// TIA Portal V16 program export: 19 tag tables, 12 data types, 33 data blocks, 85 code blocks (in call order from the OBs), 112 instance data blocks

VAR_GLOBAL   // PLC tag table "Default tag table"
   System_Byte AT %MB1 : Byte;
   FirstScan AT %M1.0 : Bool;
   DiagStatusUpdate AT %M1.1 : Bool;
   AlwaysTRUE AT %M1.2 : Bool;
   AlwaysFALSE AT %M1.3 : Bool;
   Clock_Byte AT %MB2 : Byte;
   Clock_10Hz AT %M2.0 : Bool;
   Clock_5Hz AT %M2.1 : Bool;
   "Clock_2.5Hz" AT %M2.2 : Bool;
   Clock_2Hz AT %M2.3 : Bool;
   "Clock_1.25Hz" AT %M2.4 : Bool;
   Clock_1Hz AT %M2.5 : Bool;
   "Clock_0.625Hz" AT %M2.6 : Bool;
   "Clock_0.5Hz" AT %M2.7 : Bool;
   Byte_Wekt_DRV01_R AT %MB6 : SInt;   // Bytewejściowy Status napędu
   Byte_Wekt_DRV_Temp AT %MB7 : SInt;   // Byte temp pomocniczy przy wyliczeniu wektora
   "DRV01-Bit_A/M" AT %M6.7 : Bool;   // BIt IN statusu napędu Bit Aut/manual (aut=1, manu=0)
   "DRV01-Bit_REM" AT %M6.2 : Bool;   // Bit IN statusu napędu Bit-REM Tryb aut=1 rem=0 (REM sterowanie remontowe)
   "DRV01-Bit_A" AT %M6.0 : Bool;   // Bit IN status napędu Bit-A (Alarm)
   "DRV01-Bit_Z" AT %M6.5 : Bool;   // Bit IN statusu napędu Bit-Z rozkaz załącz
   "DRV01-Bit_W" AT %M6.4 : Bool;   // Bit IN status napędu Bit-W rozkaz wyłącz
   "DRV01-Bit_R" AT %M6.6 : Bool;   // Bit IN status napędu Bit-R sygnał RESET Alarmu
   Byte_Wekt_DRV01_L AT %MB8 : Byte;   // Byte OUT wektor napędu
   Bit_DRV01_A AT %M8.0 : Bool;   // Bit OUT wektor napędu Bit-A Alarm
   Bit_DRV01_REM AT %M8.2 : Bool;   // Bit OUT wektor napędu Bit-REM tryb pracy aut=1 rem=0 (REM-sterowanie remontowe)
   Bit_DRV01_Run AT %M8.3 : Bool;   // Bit OUT wektor napędu Bit-Run (Praca stycznik załączony)
   Bit_DRV01_W AT %M8.4 : Bool;   // Bit OUT wektor napędu Bit-W rozkaz wyłącz
   Bit_DRV01_Z AT %M8.5 : Bool;   // Bit OUT wektor napędu Bit-Z rozkaz załącz
   Bit_DRV01_R AT %M8.6 : Bool;   // Bit OUT wektor napędu Bit-R ( reset alarmu)
   "Bir_DRV01_A/M" AT %M8.7 : Bool;   // Bit OUT wektor napędu Bit-A/M rodzaj pracy auto / manual (aut=1, manu=0)
   Memeory_ResAut AT %M13.2 : Bool;   // Pamięć zbocza resetu bitu automat
   apx AT %MD28 : Real;
   apx1 AT %MD32 : Real;
   apy1 AT %MD24 : Real;
   osx AT %MD50 : Real;
   osx1 AT %MD54 : Real;
   osx2 AT %MD58 : Real;
   osy AT %MD62 : Real;
   osy1 AT %MD66 : Real;
   osy2 AT %MD70 : Real;
   State_PID1 AT %MW74 : Int;
   Error_State_PID1 AT %MD76 : DWord;
   SetpointLimit_H_PID1 AT %M14.0 : Bool;   // Wartość zadanaograniczenie górnego PID1
   SetpointLimit_L_PID1 AT %M14.1 : Bool;   // Wartość zadanaograniczenie dolnego PID1
   InputWarning_H_PID1 AT %M14.2 : Bool;   // Wejście ostrzegawcze progu górnrgo PID1
   InputWarning_L_PID1 AT %M14.3 : Bool;   // Wejście ostrzegawcze progu dolnego PID1
   Reset_PID1 AT %M14.4 : Bool;   // Znacznik resetu PID1
   My_1Hz AT %M206.7 : Bool;   // Generator 1hz
   memK1 AT %M15.1 : Bool;   // Flaga pamięci K1
   pause_1 AT %M15.4 : Bool;   // Dla pomiaru nr 1 funkcji FB3
   pause_2 AT %M15.5 : Bool;   // Pałza dla pomiaru nr 2 funkcji FB3
   "Q1.1" AT %Q1.1 : Bool;
   ProcessMemory_Static_1_setChanging AT %M206.4 : Bool;   // Znacznik pobierania konfiguracji do instancji pamięci peocesu
   Tag_2 AT %MW221 : Int;
   ResetPIDManual AT %M1100.0 : Bool;   // Ręczny reset PID
   Tag_5 AT %M10101.0 : Bool;
   Reset_symulowany AT %M1040.0 : Bool;   // Pomocniczy w razie symulacji
   Tag_6 AT %M1040.5 : Bool;
   Tag_7 AT %M1040.6 : Bool;
   Tag_8 AT %M1040.7 : Bool;
   ON_OFF_AQ_Falownik AT %M1040.2 : Bool;   // Do symulacji i testów
   Sumul_OnOFF_manual_PID AT %M1100.1 : Bool;
   Symula_K2_OFF_ONN AT %M1100.3 : Bool;   // Do testów
   ResetDodtkowe AT %M1100.6 : Bool;   // Potrzeby testowe
   SymulPomoc_04 AT %M1100.4 : Bool;
   SymulPomoc_05 AT %M1100.5 : Bool;
   "I0.0" AT %I0.0 : Bool;
   "Q0.0" AT %Q0.0 : Bool;
   "Q0.1" AT %Q0.1 : Bool;
   "Q0.2" AT %Q0.2 : Bool;
   "I0.1" AT %I0.1 : Bool;
   "I0.2" AT %I0.2 : Bool;
   "I0.5" AT %I0.5 : Bool;
   "I0.6" AT %I0.6 : Bool;
   "I0.7" AT %I0.7 : Bool;
   "I1.0" AT %I1.0 : Bool;
   "I1.1" AT %I1.1 : Bool;
   "I1.2" AT %I1.2 : Bool;
   "Q0.3" AT %Q0.3 : Bool;
   "Q0.4" AT %Q0.4 : Bool;
   "Q0.5" AT %Q0.5 : Bool;
   "I0.3" AT %I0.3 : Bool;
   "I0.4" AT %I0.4 : Bool;
   "I3.7" AT %I3.7 : Bool;
   "I1.3" AT %I1.3 : Bool;
   "I1.5" AT %I1.5 : Bool;
   "I2.1" AT %I2.1 : Bool;
   "I2.0" AT %I2.0 : Bool;
   "Q1.0" AT %Q1.0 : Bool;
   "Q2.3" AT %Q2.3 : Bool;
   "Q2.2" AT %Q2.2 : Bool;
   "I1.4" AT %I1.4 : Bool;
   "Q0.6" AT %Q0.6 : Bool;
   "Q0.7" AT %Q0.7 : Bool;
   "I2.2" AT %I2.2 : Bool;
   "I2.3" AT %I2.3 : Bool;
   "I2.4" AT %I2.4 : Bool;
   "I2.5" AT %I2.5 : Bool;
   "I2.6" AT %I2.6 : Bool;
   "I2.7" AT %I2.7 : Bool;
   "I3.0" AT %I3.0 : Bool;
   "I3.1" AT %I3.1 : Bool;
   "I3.2" AT %I3.2 : Bool;
   "I3.3" AT %I3.3 : Bool;
   "I3.4" AT %I3.4 : Bool;
   "I3.5" AT %I3.5 : Bool;
   "I3.6" AT %I3.6 : Bool;
   "Q2.0" AT %Q2.0 : Bool;
   "Q2.1" AT %Q2.1 : Bool;
   "Q2.4" AT %Q2.4 : Bool;
   "Q2.5" AT %Q2.5 : Bool;
   "Q2.6" AT %Q2.6 : Bool;
   "Q2.7" AT %Q2.7 : Bool;
   "Q3.0" AT %Q3.0 : Bool;
   "Q3.1" AT %Q3.1 : Bool;
   "Q3.2" AT %Q3.2 : Bool;
   "Q3.3" AT %Q3.3 : Bool;
   "Q3.4" AT %Q3.4 : Bool;
   "Q3.5" AT %Q3.5 : Bool;
   "Q3.6" AT %Q3.6 : Bool;
   "Q3.7" AT %Q3.7 : Bool;
   "I4.0" AT %I4.0 : Bool;
   "I4.1" AT %I4.1 : Bool;
   "I4.2" AT %I4.2 : Bool;
   "I4.3" AT %I4.3 : Bool;
   "I4.4" AT %I4.4 : Bool;
   "I4.5" AT %I4.5 : Bool;
   "I4.6" AT %I4.6 : Bool;
   "I4.7" AT %I4.7 : Bool;
   "Q4.0" AT %Q4.0 : Bool;
   "Q4.1" AT %Q4.1 : Bool;
   "Q4.2" AT %Q4.2 : Bool;
   "Q4.3" AT %Q4.3 : Bool;
   "Q4.4" AT %Q4.4 : Bool;
   "Q4.5" AT %Q4.5 : Bool;
   "Q4.6" AT %Q4.6 : Bool;
   "Q4.7" AT %Q4.7 : Bool;
   Tag_3 AT %MW410 : Int;
   Tag_4 AT %MW500 : Int;
   Tag_9 AT %MW502 : Int;
   Tag_10 AT %MD500 : DWord;
   ByteH_Status_P2 AT %MB24 : Byte;   // status napędu
   ByteH_Status_P3 AT %MB26 : Byte;   // staus napędu
   ByteH_Status_P4 AT %MB28 : Byte;   // status napędu
   activePump_P1 AT %M50.4 : Bool;   // aktywna w trybie automat
   activePump_P2 AT %M50.5 : Bool;   // aktywna w trybie automat
   activePump_P3 AT %M50.6 : Bool;   // aktywna w trybie automat
   activePump_P4 AT %M50.7 : Bool;   // aktywna w trybie automat
   PV_PER_bar_modbus AT %MW400 : Int;   // Wartość bar strefa 1
   increase_O2_no1 AT %M15.6 : Bool;   // Znacznik przyrostu wartości bar 1=przyrost, 0= brak przyrostu
   "PV_PER_bar_modbus(1)" AT %MW402 : Int;   // Wartość bar strefa 2
   Tag_1 AT %M212.3 : Bool;
   stopo_dodatkow_1 AT %M15.7 : Bool;   // wyłączenie dodatkowej 1
   ris1_Hz_Calkul_bar AT %M15.2 : Bool;   // Pamięć zbocza narastającego pomiaru 1 dla funkcji FB3
   ris2_Hz_Calkul_bar AT %M15.3 : Bool;   // Pamięć zbocza narastającego nr2 dla funkcji FB3
END_VAR
VAR_GLOBAL CONSTANT   // user constants
   CONST_BUFFER_OB82 : USInt := 200;
   CONST_CUREENT2TEMPERATURE_CONVERT : Real := 50.0;
   CONST_Hz_LEVEL : Real := 33.0;
   CONST_ADC_CONVERT : Real := 27648.0;
   CONST_OUTPUT_CAREENT : Real := 20.0;
   "Local~HSC_1(2)" : Hw_Hsc := 258;
   "Local~HSC_2(2)" : Hw_Hsc := 259;
   "Local~HSC_3(2)" : Hw_Hsc := 260;
   "Local~HSC_4(2)" : Hw_Hsc := 261;
   "Local~HSC_5(2)" : Hw_Hsc := 262;
   "Local~HSC_6(2)" : Hw_Hsc := 263;
   "Local~AI2_1" : Hw_SubModule := 264;
   "Local~DI14_DQ10_1" : Hw_SubModule := 265;
   "Local~Pulse_1(2)" : Hw_Pwm := 266;
   "Local~Pulse_2(2)" : Hw_Pwm := 267;
   "Local~Pulse_3(2)" : Hw_Pwm := 268;
   "Local~Pulse_4(2)" : Hw_Pwm := 269;
   DomZabkowska : DB_WWW := 333;
   Temeratura : DB_WWW := 333;
   "Local(2)" : Hw_SubModule := 50;
   "Local~PROFINET_interface_1(2)" : Hw_Interface := 64;
   "Local~PROFINET_interface_1~Port_1(2)" : Hw_Interface := 65;
   "Local~DI_8x24VDC_1(2)" : Hw_SubModule := 270;
   OB_Main : OB_PCYCLE := 1;
   "OB_Cyclic interrupt" : OB_Cyclic := 30;
   OB_Startup : OB_STARTUP := 100;
   "Local(1)" : Hw_SubModule := 50;
   "Local~PROFINET_interface_1(1)" : Hw_Interface := 64;
   "Local~PROFINET_interface_1~Port_1(1)" : Hw_Interface := 65;
   "Local~HSC_1(1)" : Hw_Hsc := 257;
   "Local~HSC_2(1)" : Hw_Hsc := 258;
   "Local~HSC_3(1)" : Hw_Hsc := 259;
   "Local~HSC_4(1)" : Hw_Hsc := 260;
   "Local~HSC_5(1)" : Hw_Hsc := 261;
   "Local~HSC_6(1)" : Hw_Hsc := 262;
   "Local~AI_2_AQ_2_1" : Hw_SubModule := 263;
   "Local~DI_14_DQ_10_1(1)" : Hw_SubModule := 264;
   "Local~Pulse_1(1)" : Hw_Pwm := 265;
   "Local~Pulse_2(1)" : Hw_Pwm := 266;
   "Local~Pulse_3(1)" : Hw_Pwm := 267;
   "Local~Pulse_4(1)" : Hw_Pwm := 268;
   "OB_Main(1)" : OB_PCYCLE := 1;
   "Local~DI_8x24VDC_1(1)" : Hw_SubModule := 269;
   "OB_Startup(1)" : OB_STARTUP := 100;
   "~Port_2" : Hw_Interface := 66;
   "Local~AQ_4x14BIT_1(1)" : Hw_SubModule := 271;
   "~Port_2(1)" : Hw_Interface := 66;
   MS_TO_S : DInt := 1000;
   MS_TO_M : DInt := 60000;   // Pomocnicza zmienna zamiana ms na minuty
END_VAR

VAR_GLOBAL   // PLC tag table "Analogs"
   IW68 AT %IW68 : Int;
   IW66 AT %IW66 : Int;
   IW64 AT %IW64 : Int;
   IW70 AT %IW70 : Int;
   switch_kolman AT %M18.7 : Bool;   // załącz/ wyłą filtrowanie przez kolmana analogów
   "i(1)" AT %MW112 : Int;
END_VAR

VAR_GLOBAL   // PLC tag table "Error"
   Led_Error AT %M17.5 : Bool;   // Znacznik sygnalizujący wystąpienie błędu sterownika Krat
   ResetErrorOB82 AT %M17.4 : Bool;   // Znacznik resetu licznika błędów
   alarmSuchobieg AT %M93.2 : Bool;   // bit alarmu wystąpienia suchobiegu pompownia
   alarmMagistrala_niskie_bar AT %M93.3 : Bool;   // bit alarmu wystąpienia btraku ciśnienia z magistrali
   "off_AlarmMagistrala-niskie_bar" AT %M93.4 : Bool;   // bit informuje o końcu awarii magistrali niskie
   alarm_max_bar_pompownia AT %M94.0 : Bool;   // bit alarmu przekroczono max bar pompownia B7
   Discrete_alarm_18 AT %M1025.1 : Bool;   // 16#0002: Niepoprawna wartość w parametrze "Input_PER". Sprawdź, czy na wejściu analogowym występuje błąd.
   "BitMeldun-7" AT %M1029.7 : Bool;   // 16#0080: Niepoprawna wartość w trybie pracy PID. Tryb pracy nie ulega zmianie.
   Discrete_alarm_13 AT %M1024.4 : Bool;   // 16#1000: Niepoprawna wartość w parametrze "Wartość zadana": Wartość nie ma prawidłowego formatu liczbowego.
   tmp_rezerwa_1 AT %M94.1 : Bool;   // bit rezerwowy 1
   bit_off_alarm_magistrala AT %M94.2 : Bool;   // ustaw jesli koniec alarmu na magistrali bar <min
END_VAR

VAR_GLOBAL   // PLC tag table "tags"
   "Tuning.TIR_visible" AT %M1002.0 : Bool;
   "Tuning.SUT_visible" AT %M1002.1 : Bool;
   "Tuning.Mode_visible" AT %M1002.2 : Bool;
   "PID_Compact.State" AT %MW1004 : Int;
   "PID_Compact.Setpoint" AT %MD1006 : Real;
   "PID_Compact.ScaledInput" AT %MD1010 : Real;
   "PID_Compact.Output_PWM" AT %M1014.0 : Bool;
   "PID_Compact.ModeActivate" AT %M1014.1 : Bool;
   "PID_Compact.ManualEnable" AT %M1014.2 : Bool;
   "PID_Compact.Disturbance" AT %MD1016 : Real;
   "HMI.Setpoint_limited" AT %M1020.0 : Bool;
   "HMI.PhysicalUnit" AT %MB1021 : Char;
   "HMI.Output_PWM_USInt" AT %MB1022 : USInt;
   "HMI.ManualMode_visible(1)" AT %M1023.0 : Bool;
   "HMI.ManualMode_visible" AT %M1023.1 : Bool;
   "HMI.ErrorBits_Int" AT %MW1024 : Int;
   "HMI.ErrorAck_Int" AT %MW1026 : Int;
   "HMI.Warning_Int" AT %MW1028 : Int;
   "HMI.ErrorAck" AT %M1030.0 : Bool;
   "HMI.Acknowledge_visible" AT %M1030.1 : Bool;
   Communication_Alarm AT %M1030.2 : Bool;   // Znacznik błedu komunikacji HMI - PLC
   outAlarm AT %M1030.3 : Bool;   // Znacznik alarmu zbiorczego (Sygnalizator)
   "HMI.alarm_byte_1" AT %MW800 : Word;   // słowo alarmów
   "HMI.gotowość_falownik_1" AT %M800.0 : Bool;   // gotowość falownika 1
   "HMI.brak_zasilania" AT %M800.1 : Bool;   // brak zasilnia
   "HMI.SłowoStatus_Falownik1" AT %MW2000 : Int;   // Słowo statusu falownika F1
   "HMI.FalSata_bit_0" AT %M2000.0 : Bool;   // Sterowanie poprawne
   "HMI.FalSata_bit_1" AT %M2000.1 : Bool;   // falownik gotowość
   "HMI.FalSata_bit_2" AT %M2000.2 : Bool;   // wybieg
   "HMI.FalSata_bit_3" AT %M2000.3 : Bool;   // trip error
   "HMI.FalSata_bit_4" AT %M2000.4 : Bool;   // no trip error
   "HMI.FalSata_bit_5" AT %M2000.5 : Bool;   // reserved
   "HMI.FalSata_bit_6" AT %M2000.6 : Bool;   // trip zablokowany
   "HMI.FalSata_bit_7" AT %M2000.7 : Bool;   // Ostrzeżenie
   "HMI.FalSata_bit_8" AT %M2001.0 : Bool;   // prędkość = referencyjnej
   "HMI.FalSata_bit_9" AT %M2001.1 : Bool;   // listwa sterowania
   "HMI.FalSata_bit_10" AT %M2001.2 : Bool;   // częstotliwość ok
   "HMI.FalSata_bit_11" AT %M2001.3 : Bool;   // praca
   "HMI.FalSata_bit_12" AT %M2001.4 : Bool;   // rezystor hamowania
   "HMI.FalSata_bit_13" AT %M2001.5 : Bool;   // volty przekroczone
   "HMI.FalSata_bit_14" AT %M2001.6 : Bool;   // problem z momentem obrotowym
   "HMI.FalSata_bit_15" AT %M2001.7 : Bool;   // zabezpieczenie termiczne
   "HMI.kasowanie.ekranów" AT %MW1000 : Int;
   "HMI.kasowanie.ekranów_bit_0" AT %M1000.0 : Bool;   // kasowanie alarmu ekran pomp
   "HMI.kasowanie.ekranów_bit_1" AT %M1000.1 : Bool;   // kasowanie alarmu ekran zasów
   "HMI.kasowanie.ekranów_bit_2" AT %M1000.2 : Bool;
   "HMI.kasowanie.ekranów_bit_3" AT %M1000.3 : Bool;
   "HMI.kasowanie.ekranów_bit_4" AT %M1000.4 : Bool;
   "HMI.kasowanie.ekranów_bit_5" AT %M1000.5 : Bool;
   "HMI.kasowanie.ekranów_bit_6" AT %M1000.6 : Bool;
   "HMI.kasowanie.ekranów_bit_7" AT %M1000.7 : Bool;
   "HMI.alarm_01" AT %M1001.0 : Bool;   // Alarm Modbus RTU
   "HMI.alarm_02" AT %M1001.1 : Bool;   // Ostrzerzenie Modbus RTU
   "HMI.alarm_01(2)" AT %M1001.2 : Bool;
   "HMI.alarm_01(3)" AT %M1001.3 : Bool;
   "HMI.alarm_01(4)" AT %M1001.4 : Bool;
   "HMI.alarm_01(5)" AT %M1001.5 : Bool;
   "HMI.alarm_01(6)" AT %M1001.6 : Bool;
   "HMI.alarm_01(7)" AT %M1001.7 : Bool;
END_VAR

VAR_GLOBAL   // PLC tag table "MP04_1"
   temp_current_fow_H_Q1 AT %MW600 : Word;   // H byte przepływ aktualny VF
   tmp_current_fow_L_Q1 AT %MW602 : Word;   // L byte przepływ aktualny VF
   tmp_front_volumeVF_H_Q1 AT %MW604 : Word;   // licznik objetości przód H byte
   tmp_front_volumeVF_L_Q1 AT %MW606 : Word;   // licznik objetości przód L byte
   tmp_back_balueVR_H_Q1 AT %MW608 : Word;   // licznik objętości wstecz H byte
   tmp_back_balueVR_L_Q1 AT %MW610 : Word;   // licznik objętości wstecz L byte
   "tmp_differential counter VD_H_Q1" AT %MW612 : Word;   // licznik różnicowy VD H byte
   "tmp_differential counter VD_L_Q1" AT %MW614 : Word;   // licznik różnicowy VD L byte
   "tmp_volume counter status _GF_H_Q1" AT %MW616 : Word;   // statu licznik objetości GF H byte
   "tmp_volume counter status _GF_L_Q1" AT %MW618 : Word;   // status licznik objetości GF L byte
   "tmp_volume counter status_GR_H_Q1" AT %MW620 : Word;   // statu licznik objetości GR H byte
   "tmp_volume counter status_GR_L_Q1" AT %MW622 : Word;   // statu licznik objetości GR L byte
   "tmp_differential counter status_GD_H_Q1" AT %MW624 : Word;   // statu licznik objetości GD H byte
   "tmp_differential counter status_GD_L_Q1" AT %MW626 : Word;   // statu licznik objetości GD L byte
   tmp_sataus_MP04_Q1 AT %MW628 : Word;   // staus urządzenia MP04_Q1
   temp_current_fow_H_Q2 AT %MW630 : Word;   // H byte przepływ aktualny VF
   tmp_current_fow_L_Q2 AT %MW632 : Word;   // L byte przepływ aktualny VF
   tmp_front_volumeVF_H_Q2 AT %MW634 : Word;   // licznik objetości przód H byte
   tmp_front_volumeVF_L_Q2 AT %MW636 : Word;   // licznik objetości przód L byte
   tmp_back_balueVR_H_Q2 AT %MW638 : Word;   // licznik objętości wstecz H byte
   tmp_back_balueVR_L_Q2 AT %MW640 : Word;   // licznik objętości wstecz L byte
   "tmp_differential counter VD_H_Q2" AT %MW642 : Word;   // licznik różnicowy VD H byte
   "tmp_differential counter VD_L_Q2" AT %MW644 : Word;   // licznik różnicowy VD L byte
   "tmp_volume counter status _GF_H_Q2" AT %MW646 : Word;   // statu licznik objetości GF H byte
   "tmp_volume counter status _GF_L_Q2" AT %MW648 : Word;   // status licznik objetości GF L byte
   "tmp_volume counter status_GR_H_Q2" AT %MW650 : Word;   // statu licznik objetości GR H byte
   "tmp_volume counter status_GR_L_Q2" AT %MW652 : Word;   // statu licznik objetości GR L byte
   "tmp_differential counter status_GD_H_Q2" AT %MW654 : Word;   // statu licznik objetości GD H byte
   "tmp_differential counter status_GD_L_Q2" AT %MW656 : Word;   // statu licznik objetości GD L byte
   tmp_sataus_MP04_Q2 AT %MW658 : Word;   // staus urządzenia MP04_Q2
END_VAR

VAR_GLOBAL   // PLC tag table "ModbusRTU"
   setErrorModbsmasterFal AT %M18.0 : Bool;   // error bit modbus master falownik / Znacznik błedu komunikacji modbus
   setErrorModbsmasterMPP04_1 AT %M18.1 : Bool;   // error bit modbus master przepływomierz / Znacznik błedu komunikacji modbus
   setErrorModbsSlave AT %M18.2 : Bool;   // error bit modbus slave / Znacznik błedu komunikacji modbus
   "setErrorModbs----" AT %M18.3 : Bool;   // Znacznik błedu komunikacji modbus
   memRisErrorModbusmaster AT %M16.6 : Bool;   // Pamięć zbocza błędu komunikacji
   memReisModbus_Loop1 AT %M16.2 : Bool;   // Znacznik pamięci zbocza dla pętli 1
   memRisModbusmaster_Loop2 AT %M16.3 : Bool;   // pamięć zbocza dla petli 2 modbas
   memRisModbusmaster_Loop3 AT %M16.4 : Bool;   // pamięć zbocza pętli 3 modbas
   memRisModbus_Loop AT %M16.5 : Bool;   // Pamieć zbocza do uruchomienia petli SC1000
   ndrSlave AT %M16.7 : Bool;   // bit nowe dane gotowe / Pamieć zbocza błedu komunikacji
   drSlave AT %M14.5 : Bool;   // bit czytanie danych / pamięć zbocza błędu komunikacji
   memRisErrorModbusMPP04_1 AT %M14.6 : Bool;   // pamięć zbocza error modbus MPP04-1
   StatusSlave AT %MW29 : Word;   // Status slave Modbus RTU
   errorSatausSlave AT %MW31 : Word;   // Status błędu slave Modbus RTU
   setErrorModbsmasterMPP04_2 AT %M93.0 : Bool;   // error bit modbus master przepływomierz / Znacznik błedu komunikacji modbus
   memRisErrorModbusMPP04_2 AT %M14.7 : Bool;   // pamięć zbocza error modbus MPP04-1
   memRisErrorModbusFal AT %M93.1 : Bool;   // pamięć zbocza error modbus MPP04-1
   "memStep_errorMPP04-1" AT %MB100 : USInt;   // bajt pamieci w którym kroku nastąpił błąd modbus
   "memStep_errorMPP04-2" AT %MB101 : USInt;   // bajt pamieci w którym kroku nastąpił błąd modbus
   memStep_errorFal AT %MB102 : USInt;   // bajt pamieci w którym kroku nastąpił błąd modbus
   memStep_errorSlave AT %MB103 : USInt;   // bajt pamieci w którym kroku nastąpił błąd modbus
   "memRisSteperror_MPP04-1" AT %M104.0 : Bool;   // pamięć zbocza dla przechwycenia kroku błedu
   "memRisSteperror_MPP04-2" AT %M104.1 : Bool;   // pamięć zbocza dla przechwycenia kroku błedu
   memRisSteperror_Fal AT %M104.2 : Bool;   // pamięć zbocza dla przechwycenia kroku błedu
   memRisSteperror AT %M104.3 : Bool;   // pamięć zbocza dla przechwycenia kroku błedu
   act_flow_Q1 AT %MD600 : DWord;   // wartość przepływu Q1
   act_front_volumeVF_Q1 AT %MD604 : DWord;   // licznik objetości przód Q1
   act_back_valueVR_Q1 AT %MD608 : DWord;   // licznika objętości w tył Q1
   "act_differential counter VD_Q1" AT %MD612 : DWord;   // liczni różnicowyobjętości VD Q1
   "act_volume counter status _GF_Q1" AT %MD616 : DWord;   // główny licznik objetosci przód GF Q1
   "act_volume counter status_GR_Q1" AT %MD620 : DWord;   // główny licznik objetości w tył GR Q1
   "act_differential counter status_GD_Q1" AT %MD624 : DWord;   // główny różnicow licznik objetości GD Q1
   act_flow_Q2 AT %MD630 : DWord;   // wartość przepływu Q2
   act_ValueVF_Q2 AT %MD634 : DWord;   // licznik objetości przód Q2
   act_front_volumeVF_Q2 AT %MD638 : DWord;   // licznika objętości w tył Q2
   act_back_balueVR_Q2 AT %MD642 : DWord;   // liczni różnicowyobjętości VD Q2
   "act_differential counter VD_Q2" AT %MD646 : DWord;   // główny licznik objetosci przód GF Q2
   "act_volume counter status _GF_Q2" AT %MD650 : DWord;   // główny licznik objetości w tył GR Q2
   "act_volume counter status_GR_Q2" AT %MD654 : DWord;   // główny różnicow licznik objetości GD Q2
   "act_differential counter status_GD_Q2" AT %MD658 : DWord;
   Switch_PrzepłtwSygnał AT %M92.0 : Bool;   // wybór źródła wartości pomiaru analog / modbus rtu
END_VAR

VAR_GLOBAL   // PLC tag table "ModbusTCP"
   memTrgServer_1 AT %M106.0 : Bool;
   memTrgServer_2 AT %M106.1 : Bool;
   memTrgServer_3 AT %M106.2 : Bool;
   DISCONNECT_SERVER_1 AT %M106.3 : Bool;
   DISCONNECT_SERVER_2 AT %M106.4 : Bool;
   DISCONNECT_SERVER_3 AT %M106.5 : Bool;
   memRisingTriger_Data_4 AT %M107.1 : Bool;   // pamieć zbocza narastającego przekazania danej do wysłania
   memRisingTriger_Data_11 AT %M108.0 : Bool;   // pamieć zbocza narastającego przekazania danej do wysłania
   memRisingTriger_Data_5 AT %M107.2 : Bool;   // pamieć zbocza narastającego przekazania danej do wysłania
   memRisingTriger_Data_8 AT %M107.5 : Bool;   // pamieć zbocza narastającego przekazania danej do wysłania
   memRisingTriger_Data_1 AT %M106.6 : Bool;   // pamieć zbocza narastającego przekazania danej do wysłania
   memRisingTriger_Data_13 AT %M108.2 : Bool;   // pamieć zbocza narastającego przekazania danej do wysłania
   memRisingTriger_Data_2 AT %M106.7 : Bool;   // pamieć zbocza narastającego przekazania danej do wysłania
   memRisingTriger_Data_6 AT %M107.3 : Bool;   // pamieć zbocza narastającego przekazania danej do wysłania
   memRisingTriger_Data_10 AT %M107.7 : Bool;   // pamieć zbocza narastającego przekazania danej do wysłania
   memRisingTriger_Data_12 AT %M108.1 : Bool;   // pamieć zbocza narastającego przekazania danej do wysłania
   memRisingTriger_Data_3 AT %M107.0 : Bool;   // pamieć zbocza narastającego przekazania danej do wysłania
   memRisingTriger_Data_9 AT %M107.6 : Bool;   // pamieć zbocza narastającego przekazania danej do wysłania
   memRisingTriger_Data_7 AT %M107.4 : Bool;   // pamieć zbocza narastającego przekazania danej do wysłania
   DISCONNECT_SERVER_4 AT %M108.3 : Bool;
   memTrgServer_4 AT %M108.4 : Bool;
   memTrig_Client_Receiving_16 AT %M110.4 : Bool;
   memTrig_Client_Receiving_7 AT %M109.3 : Bool;
   memTrig_Client_Receiving_11 AT %M109.7 : Bool;
   memRisingTriger_Data_1_2 AT %M110.6 : Bool;   // pamieć zbocza narastającego przekazania danej do wysłania
   memRisingTriger_Data_1_1 AT %M110.5 : Bool;   // pamieć zbocza narastającego przekazania danej do wysłania
   memTrig_Client_Receiving_5 AT %M109.1 : Bool;
   memTrig_Client_Receiving_13 AT %M110.1 : Bool;
   memTrig_Client_Receiving_14 AT %M110.2 : Bool;
   memTrig_Client_Receiving_3 AT %M108.7 : Bool;
   memTrig_Client_Receiving_8 AT %M109.4 : Bool;
   memTrig_Client_Receiving_10 AT %M109.6 : Bool;
   memTrig_Client_Receiving_6 AT %M109.2 : Bool;
   memTrig_Client_Receiving_12 AT %M110.0 : Bool;
   memTrig_Client_Receiving_2 AT %M108.6 : Bool;
   memTrig_Client_Receiving_1 AT %M108.5 : Bool;
   memTrig_Client_Receiving_4 AT %M109.0 : Bool;
   memTrig_Client_Receiving_9 AT %M109.5 : Bool;
   memTrig_Client_Receiving_15 AT %M110.3 : Bool;
   memRisingTriger_Data_16 AT %M111.2 : Bool;
   memRisingTriger_Data_14 AT %M111.0 : Bool;
   memRisingTriger_Data_15 AT %M111.1 : Bool;
   memRisingTriger_Data_47 AT %M115.1 : Bool;
   memTrig_Client_Receiving_17 AT %M120.2 : Bool;
   memTrig_Client_Receiving_87 AT %M129.0 : Bool;
   memTrig_Client_Receiving_23 AT %M121.0 : Bool;
   memRisingTriger_Data_29 AT %M112.7 : Bool;
   memTrig_Client_Receiving_84 AT %M128.5 : Bool;
   memTrig_Client_Receiving_43 AT %M123.4 : Bool;
   memRisingTriger_Data_63 AT %M117.1 : Bool;
   memTrig_Client_Receiving_74 AT %M127.3 : Bool;
   memRisingTriger_Data_69 AT %M117.7 : Bool;
   memRisingTriger_Data_70 AT %M118.0 : Bool;
   memTrig_Client_Receiving_32 AT %M122.1 : Bool;
   memRisingTriger_Data_80 AT %M119.2 : Bool;
   memTrig_Client_Receiving_65 AT %M126.2 : Bool;
   memTrig_Client_Receiving_71 AT %M127.0 : Bool;
   memTrig_Client_Receiving_36 AT %M122.5 : Bool;
   memRisingTriger_Data_84 AT %M119.6 : Bool;
   memRisingTriger_Data_68 AT %M117.6 : Bool;
   memTrig_Client_Receiving_49 AT %M124.2 : Bool;
   memRisingTriger_Data_85 AT %M119.7 : Bool;
   memRisingTriger_Data_36 AT %M113.6 : Bool;
   memTrig_Client_Receiving_76 AT %M127.5 : Bool;
   memTrig_Client_Receiving_70 AT %M126.7 : Bool;
   memTrig_Client_Receiving_89 AT %M129.2 : Bool;
   memRisingTriger_Data_19 AT %M111.5 : Bool;
   memRisingTriger_Data_31 AT %M113.1 : Bool;
   memTrig_Client_Receiving_20 AT %M120.5 : Bool;
   memTrig_Client_Receiving_48 AT %M124.1 : Bool;
   memTrig_Client_Receiving_56 AT %M125.1 : Bool;
   memRisingTriger_Data_44 AT %M114.6 : Bool;
   memTrig_Client_Receiving_82 AT %M128.3 : Bool;
   memTrig_Client_Receiving_58 AT %M125.3 : Bool;
   memTrig_Client_Receiving_67 AT %M126.4 : Bool;
   memRisingTriger_Data_57 AT %M116.3 : Bool;
   memTrig_Client_Receiving_80 AT %M128.1 : Bool;
   memRisingTriger_Data_52 AT %M115.6 : Bool;
   memTrig_Client_Receiving_69 AT %M126.6 : Bool;
   memRisingTriger_Data_64 AT %M117.2 : Bool;
   memTrig_Client_Receiving_60 AT %M125.5 : Bool;
   memTrig_Client_Receiving_62 AT %M125.7 : Bool;
   memRisingTriger_Data_26 AT %M112.4 : Bool;
   memRisingTriger_Data_82 AT %M119.4 : Bool;
   memRisingTriger_Data_72 AT %M118.2 : Bool;
   memTrig_Client_Receiving_26 AT %M121.3 : Bool;
   memRisingTriger_Data_73 AT %M118.3 : Bool;
   memRisingTriger_Data_46 AT %M115.0 : Bool;
   memTrig_Client_Receiving_73 AT %M127.2 : Bool;
   memTrig_Client_Receiving_24 AT %M121.1 : Bool;
   memRisingTriger_Data_42 AT %M114.4 : Bool;
   memTrig_Client_Receiving_78 AT %M127.7 : Bool;
   memRisingTriger_Data_27 AT %M112.5 : Bool;
   memTrig_Client_Receiving_25 AT %M121.2 : Bool;
   memRisingTriger_Data_34 AT %M113.4 : Bool;
   memTrig_Client_Receiving_30 AT %M121.7 : Bool;
   memTrig_Client_Receiving_47 AT %M124.0 : Bool;
   memRisingTriger_Data_71 AT %M118.1 : Bool;
   memRisingTriger_Data_18 AT %M111.4 : Bool;
   memRisingTriger_Data_33 AT %M113.3 : Bool;
   memTrig_Client_Receiving_85 AT %M128.6 : Bool;
   memRisingTriger_Data_17 AT %M111.3 : Bool;
   memRisingTriger_Data_74 AT %M118.4 : Bool;
   memRisingTriger_Data_35 AT %M113.5 : Bool;
   memTrig_Client_Receiving_42 AT %M123.3 : Bool;
   memTrig_Client_Receiving_37 AT %M122.6 : Bool;
   memTrig_Client_Receiving_22 AT %M120.7 : Bool;
   memRisingTriger_Data_81 AT %M119.3 : Bool;
   memTrig_Client_Receiving_18 AT %M120.3 : Bool;
   memRisingTriger_Data_87 AT %M120.1 : Bool;
   memRisingTriger_Data_62 AT %M117.0 : Bool;
   memTrig_Client_Receiving_19 AT %M120.4 : Bool;
   memRisingTriger_Data_40 AT %M114.2 : Bool;
   memTrig_Client_Receiving_46 AT %M123.7 : Bool;
   memTrig_Client_Receiving_63 AT %M126.0 : Bool;
   memTrig_Client_Receiving_35 AT %M122.4 : Bool;
   memRisingTriger_Data_83 AT %M119.5 : Bool;
   memTrig_Client_Receiving_21 AT %M120.6 : Bool;
   memTrig_Client_Receiving_83 AT %M128.4 : Bool;
   memRisingTriger_Data_39 AT %M114.1 : Bool;
   memRisingTriger_Data_53 AT %M115.7 : Bool;
   memTrig_Client_Receiving_44 AT %M123.5 : Bool;
   memRisingTriger_Data_45 AT %M114.7 : Bool;
   memRisingTriger_Data_37 AT %M113.7 : Bool;
   memTrig_Client_Receiving_38 AT %M122.7 : Bool;
   memTrig_Client_Receiving_79 AT %M128.0 : Bool;
   memRisingTriger_Data_32 AT %M113.2 : Bool;
   memRisingTriger_Data_22 AT %M112.0 : Bool;
   memTrig_Client_Receiving_72 AT %M127.1 : Bool;
   memTrig_Client_Receiving_31 AT %M122.0 : Bool;
   memTrig_Client_Receiving_68 AT %M126.5 : Bool;
   memTrig_Client_Receiving_55 AT %M125.0 : Bool;
   memRisingTriger_Data_67 AT %M117.5 : Bool;
   memRisingTriger_Data_41 AT %M114.3 : Bool;
   memRisingTriger_Data_28 AT %M112.6 : Bool;
   memRisingTriger_Data_61 AT %M116.7 : Bool;
   memTrig_Client_Receiving_64 AT %M126.1 : Bool;
   memTrig_Client_Receiving_50 AT %M124.3 : Bool;
   memRisingTriger_Data_76 AT %M118.6 : Bool;
   memRisingTriger_Data_30 AT %M113.0 : Bool;
   memRisingTriger_Data_58 AT %M116.4 : Bool;
   memRisingTriger_Data_75 AT %M118.5 : Bool;
   memRisingTriger_Data_60 AT %M116.6 : Bool;
   memRisingTriger_Data_56 AT %M116.2 : Bool;
   memTrig_Client_Receiving_34 AT %M122.3 : Bool;
   memTrig_Client_Receiving_52 AT %M124.5 : Bool;
   memTrig_Client_Receiving_27 AT %M121.4 : Bool;
   memRisingTriger_Data_54 AT %M116.0 : Bool;
   memRisingTriger_Data_25 AT %M112.3 : Bool;
   memTrig_Client_Receiving_33 AT %M122.2 : Bool;
   memRisingTriger_Data_23 AT %M112.1 : Bool;
   memRisingTriger_Data_66 AT %M117.4 : Bool;
   memTrig_Client_Receiving_88 AT %M129.1 : Bool;
   memRisingTriger_Data_51 AT %M115.5 : Bool;
   memRisingTriger_Data_43 AT %M114.5 : Bool;
   memRisingTriger_Data_86 AT %M120.0 : Bool;
   memRisingTriger_Data_65 AT %M117.3 : Bool;
   memTrig_Client_Receiving_66 AT %M126.3 : Bool;
   memTrig_Client_Receiving_28 AT %M121.5 : Bool;
   memTrig_Client_Receiving_51 AT %M124.4 : Bool;
   memTrig_Client_Receiving_59 AT %M125.4 : Bool;
   memRisingTriger_Data_38 AT %M114.0 : Bool;
   memTrig_Client_Receiving_45 AT %M123.6 : Bool;
   memRisingTriger_Data_79 AT %M119.1 : Bool;
   memTrig_Client_Receiving_81 AT %M128.2 : Bool;
   memRisingTriger_Data_50 AT %M115.4 : Bool;
   memTrig_Client_Receiving_86 AT %M128.7 : Bool;
   memRisingTriger_Data_55 AT %M116.1 : Bool;
   memTrig_Client_Receiving_41 AT %M123.2 : Bool;
   memTrig_Client_Receiving_54 AT %M124.7 : Bool;
   memRisingTriger_Data_49 AT %M115.3 : Bool;
   memTrig_Client_Receiving_53 AT %M124.6 : Bool;
   memTrig_Client_Receiving_61 AT %M125.6 : Bool;
   memRisingTriger_Data_59 AT %M116.5 : Bool;
   memTrig_Client_Receiving_77 AT %M127.6 : Bool;
   memTrig_Client_Receiving_29 AT %M121.6 : Bool;
   memRisingTriger_Data_77 AT %M118.7 : Bool;
   memRisingTriger_Data_48 AT %M115.2 : Bool;
   memTrig_Client_Receiving_40 AT %M123.1 : Bool;
   memRisingTriger_Data_24 AT %M112.2 : Bool;
   memTrig_Client_Receiving_57 AT %M125.2 : Bool;
   memRisingTriger_Data_20 AT %M111.6 : Bool;
   timeDISCONECT_TCP_SERVER_1 AT %M111.7 : Bool;
   timeDISCONECT_TCP_SERVER_2 AT %M123.0 : Bool;
   timeDISCONECT_TCP_SERVER_3 AT %M119.0 : Bool;
   timeDISCONECT_TCP_SERVER_4 AT %M127.4 : Bool;
END_VAR

VAR_GLOBAL   // PLC tag table "P1"
   inputReadyP1 AT %M81.4 : Bool;   // sugnał gotowość / Gotowość napędu
   inputRunF_P1 AT %M81.5 : Bool;   // stycznik falownik / Potwierdzenie pracy z falownika
   inputRunS_P1 AT %M81.6 : Bool;   // stycznik softstart / Powierdzenie pracy z sieci
   CMD_inverter_P1 AT %M81.7 : Bool;   // Stycznik Falownik
   CMD_network_P1 AT %M82.0 : Bool;   // Stycznik Sieć
   setCMD_FP1 AT %M207.0 : Bool;   // Znacznik sterowania w trybie falownik dlaP1
   setCMD_SP1 AT %M207.1 : Bool;   // Znacznik sterowania w trybie sieć
   IsReady_P1 AT %M17.0 : Bool;   // Znacznik gotowości napędu
   Hour_Work_P1 AT %MD36 : DWord;   // Licznik pracy
   Set_HWork_P1 AT %M19.0 : Bool;   // Znacznik ustawienia aktywnej do pracy (po porównaniu liczników pracy)
   IsRunInverter_P1 AT %M211.3 : Bool;   // Potwierdzenie pracy z falownika
   IsRunNetwork_P1 AT %M217.0 : Bool;   // Potwierdzenie pracy z sieci
   Is_extras_K1_P1 AT %M218.4 : Bool;   // Znacznik motor dodatkowy nr 1
   setSUPV_FP1 AT %M12.0 : Bool;   // Znacznik polecenia startu z falownika
   IsRun_P1 AT %M10.4 : Bool;   // Potwierdzenie pracy
   setSUPV_SP1 AT %M12.7 : Bool;   // Znacznik polecenia startu z sieci
   "Ustaw alarm P1" AT %M1040.1 : Bool;   // symulacyjny bit alarmu
   CMD_soft_P1 AT %M84.7 : Bool;   // sygnał z softstart potwierdzenie pracy / sygnał on/off soft-start
   CB_CMD_P1 AT %M12.4 : Bool;   // Znacznik polecenia on/off przekaźnik napędu
   resetFault_SoftStart_P1 AT %M50.0 : Bool;   // sygnał resetu softstart
   bitH_Alarm_P1 AT %M22.0 : Bool;   // Alarm - kopia bitu z instancji statusu napędu
   bitH_REM_P1 AT %M22.2 : Bool;   // Zdalna - kopia bitu z instancji statusu napędu
   bitH_RUN_P1 AT %M22.3 : Bool;   // Praca - kopia bitu z instancji statusu napędu
   bitH_OFF_P1 AT %M22.4 : Bool;   // Polecenie OFF - kopia bitu z instancji statusu napędu
   bitH_ON_P1 AT %M22.5 : Bool;   // Polecenie ON - kopia bitu z instancji statusu napędu
   bitH_Res_P1 AT %M22.6 : Bool;   // Reset - kopia bitu z instancji statusu napędu
   bitH_Aut_Man_P1 AT %M22.7 : Bool;   // Aut=1 Man=0 - kopia bitu z instancji statusu napędu
   Is_extras_K3_P1 AT %M17.7 : Bool;   // Znacznik motor dodatkowy nr 3
   Is_extras_K2_P1 AT %M218.7 : Bool;   // Znacznik motor dodatkowy nr 2
   off_add_K1_P1 AT %M52.0 : Bool;   // sterowanie wyłączeniem selektywnym dodatkowej
   off_add_K2_P1 AT %M52.1 : Bool;   // sterowanie wyłączeniem selektywnym dodatkowej
   off_add_K3_P1 AT %M52.2 : Bool;   // sterowanie wyłączeniem selektywnym dodatkowej
   off_add_K4_P1 AT %M53.4 : Bool;   // sterowanie wyłączeniem selektywnym dodatkowej
   Set_50Hz_M AT %M217.6 : Bool;   // Znacznik pamięci podtrzymujący przełączenie na sieć
   Mem_Res_setCMD_MC_P1 AT %M223.0 : Bool;   // pamięć zbocza załączenia timera blokowania stycznika falowni
   CMD_ErrorSet_NetworkP1 AT %M221.3 : Bool;   // Znacznik sterowania awaryjnego pracą pompy bez falownika
END_VAR

VAR_GLOBAL   // PLC tag table "P2"
   inputReadyP2 AT %M82.1 : Bool;   // sugnał gotowość / Gotowość napędu
   inputRunF_P2 AT %M82.2 : Bool;   // stycznik falownik / Potwierdzenie pracy z falownika
   inputRunS_P2 AT %M82.3 : Bool;   // stycznik softstart / Powierdzenie pracy z sieci
   CMD_inverter_P2 AT %M82.4 : Bool;   // Stycznik Falownik
   CMD_network_P2 AT %M82.5 : Bool;   // Stycznik Sieć
   setCMD_FP2 AT %M207.2 : Bool;   // Znacznik sterowania w trybie falownik dlaP1
   setCMD_SP2 AT %M207.3 : Bool;   // Znacznik sterowania w trybie sieć
   IsReady_P2 AT %M17.1 : Bool;   // Znacznik gotowości napędu
   CB_CMD_P2 AT %M12.5 : Bool;   // Znacznik polecenia on/off przekaźnik napędu
   Set_HWork_P2 AT %M11.1 : Bool;   // Znacznik ustawienia aktywnej do pracy (po porównaniu liczników pracy)
   IsRunInverter_P2 AT %M211.4 : Bool;   // Potwierdzenie pracy z falownika
   IsRunNetwork_P2 AT %M217.1 : Bool;   // Potwierdzenie pracy z sieci
   Is_extras_K1_P2 AT %M218.5 : Bool;   // Znacznik motor dodatkowy nr 1
   setSUPV_FP2 AT %M12.1 : Bool;   // Znacznik polecenia startu z falownika
   IsRun_P2 AT %M10.5 : Bool;   // Potwierdzenie pracy
   setSUPV_SP2 AT %M13.0 : Bool;   // Znacznik polecenia startu z sieci
   CMD_soft_P2 AT %M85.0 : Bool;   // sygnał z softstart potwierdzenie pracy / sygnał on/off soft-start
   resetFault_SoftStart_P2 AT %M50.1 : Bool;   // sygnał resetu softstart
   bitH_Alarm_P2 AT %M24.0 : Bool;   // Alarm - kopia bitu z instancji statusu napędu
   bitH_REM_P2 AT %M24.2 : Bool;   // Zdalna - kopia bitu z instancji statusu napędu
   bitH_RUN_P2 AT %M24.3 : Bool;   // Praca - kopia bitu z instancji statusu napędu
   bitH_OFF_P2 AT %M24.4 : Bool;   // Polecenie OFF - kopia bitu z instancji statusu napędu
   bitH_ON_P2 AT %M24.5 : Bool;   // Polecenie ON - kopia bitu z instancji statusu napędu
   bitH_Res_P2 AT %M24.6 : Bool;   // Reset - kopia bitu z instancji statusu napędu
   bitH_Aut_Man_P2 AT %M24.7 : Bool;   // Aut=1 Man=0 - kopia bitu z instancji statusu napędu
   bitH_rezerwa_P2 AT %M24.1 : Bool;   // rez
   Is_extras_K3_P2 AT %M89.6 : Bool;   // Znacznik motor dodatkowy nr 3
   Is_extras_K2_P2 AT %M219.0 : Bool;   // Znacznik motor dodatkowy nr 2
   off_add_K1_P2 AT %M52.3 : Bool;   // sterowanie wyłączeniem selektywnym dodatkowej
   off_add_K2_P2 AT %M52.4 : Bool;   // sterowanie wyłączeniem selektywnym dodatkowej
   off_add_K3_P2 AT %M52.5 : Bool;   // sterowanie wyłączeniem selektywnym dodatkowej
   off_add_K4_P2 AT %M53.5 : Bool;   // sterowanie wyłączeniem selektywnym dodatkowej
   CMD_ErrorSet_NetworkP2 AT %M221.4 : Bool;   // Znacznik sterowania awaryjnego pracą pompy bez falownika
   Hour_Work_P2 AT %MD40 : DWord;   // Licznik pracy
   "Ustaw alarm P2" AT %M1040.3 : Bool;   // symulacyjny bit alarmu
   Set_50Hz_P2 AT %M217.7 : Bool;   // Znacznik pamięci podtrzymujący przełączenie na sieć
   Mem_Res_setCMD_MC_P2 AT %M223.1 : Bool;   // pamięć zbocza załączenia timera blokowania stycznika falowni
END_VAR

VAR_GLOBAL   // PLC tag table "P3"
   inputReadyP3 AT %M82.6 : Bool;   // sugnał gotowość / Gotowość napędu
   inputRunF_P3 AT %M82.7 : Bool;   // stycznik falownik / Potwierdzenie pracy z falownika
   inputRunS_P3 AT %M83.0 : Bool;   // stycznik softstart / Powierdzenie pracy z sieci
   CMD_inverter_P3 AT %M83.1 : Bool;   // Stycznik Falownik
   CMD_network_P3 AT %M83.2 : Bool;   // Stycznik Sieć
   setCMD_FP3 AT %M207.4 : Bool;   // Znacznik sterowania w trybie falownik dlaP1
   setCMD_SP3 AT %M207.5 : Bool;   // Znacznik sterowania w trybie sieć
   IsReady_P3 AT %M17.2 : Bool;   // Znacznik gotowości napędu
   CB_CMD_P3 AT %M12.6 : Bool;   // Znacznik polecenia on/off przekaźnik napędu
   Hour_Work_P3 AT %MD44 : DWord;   // Licznik pracy
   Set_HWork_P3 AT %M11.2 : Bool;   // Znacznik ustawienia aktywnej do pracy (po porównaniu liczników pracy)
   IsRunInverter_P3 AT %M211.5 : Bool;   // Potwierdzenie pracy z falownika
   IsRunNetwork_P3 AT %M217.2 : Bool;   // Potwierdzenie pracy z sieci
   Is_extras_K1_P3 AT %M218.6 : Bool;   // Znacznik motor dodatkowy nr 1
   Set_50Hz_P3 AT %M219.5 : Bool;   // Znacznik pamięci podtrzymujący przełączenie na sieć
   setSUPV_FP3 AT %M12.2 : Bool;   // Znacznik polecenia startu z falownika
   IsRun_P3 AT %M11.6 : Bool;   // Potwierdzenie pracy
   setSUPV_SP3 AT %M13.1 : Bool;   // Znacznik polecenia startu z sieci
   CMD_soft_P3 AT %M85.1 : Bool;   // sygnał z softstart potwierdzenie pracy / sygnał on/off soft-start
   resetFault_SoftStart_P3 AT %M50.2 : Bool;   // sygnał resetu softstart
   bitH_REM_P3 AT %M26.2 : Bool;   // Zdalna - kopia bitu z instancji statusu napędu
   bitH_RUN_P3 AT %M26.3 : Bool;   // Praca - kopia bitu z instancji statusu napędu
   bitH_OFF_P3 AT %M26.4 : Bool;   // Polecenie OFF - kopia bitu z instancji statusu napędu
   bitH_ON_P3 AT %M26.5 : Bool;   // Polecenie ON - kopia bitu z instancji statusu napędu
   bitH_Res_P3 AT %M26.6 : Bool;   // Reset - kopia bitu z instancji statusu napędu
   bitH_Aut_Man_P3 AT %M26.7 : Bool;   // Aut=1 Man=0 - kopia bitu z instancji statusu napędu
   bitH_Alarm_P3 AT %M26.0 : Bool;   // Alarm - kopia bitu z instancji statusu napędu
   bitH_rezerwa_P3 AT %M26.1 : Bool;   // rez
   Is_extras_K3_P3 AT %M89.7 : Bool;   // Znacznik motor dodatkowy nr 3
   Is_extras_K2_P3 AT %M219.1 : Bool;   // Znacznik motor dodatkowy nr 2
   off_add_K1_P3 AT %M52.6 : Bool;   // sterowanie wyłączeniem selektywnym dodatkowej
   off_add_K2_P3 AT %M52.7 : Bool;   // sterowanie wyłączeniem selektywnym dodatkowej
   off_add_K3_P3 AT %M53.0 : Bool;   // sterowanie wyłączeniem selektywnym dodatkowej
   off_add_K4_P3 AT %M53.6 : Bool;   // sterowanie wyłączeniem selektywnym dodatkowej
   CMD_ErrorSet_NetworkM3 AT %M221.5 : Bool;   // Znacznik sterowania awaryjnego pracą pompy bez falownika
   Mem_Res_setCMD_MC_P3 AT %M223.2 : Bool;   // pamięć zbocza załączenia timera blokowania stycznika falowni
END_VAR

VAR_GLOBAL   // PLC tag table "P4"
   inputRunF_P4 AT %M81.3 : Bool;   // stycznik falownik / Potwierdzenie pracy z falownika
   inputRunS_P4 AT %M80.7 : Bool;   // stycznik softstart / Powierdzenie pracy z sieci
   inputReadyP4 AT %M80.3 : Bool;   // sugnał gotowość / Gotowość napędu
   IsReady_P4 AT %M83.3 : Bool;   // Znacznik gotowości napędu
   IsRunInverter_P4 AT %M83.4 : Bool;   // Potwierdzenie pracy z falownika
   IsRunNetwork_P4 AT %M83.5 : Bool;   // Potwierdzenie pracy z sieci
   CMD_inverter_P4 AT %M83.6 : Bool;   // Stycznik Falownik
   CMD_network_P4 AT %M83.7 : Bool;   // Stycznik Sieć
   CMD_soft_P4 AT %M85.2 : Bool;   // sygnał z softstart potwierdzenie pracy / sygnał on/off soft-start
   setCMD_FP4 AT %M87.0 : Bool;   // Znacznik sterowania w trybie falownik dlaP1
   setCMD_SP4 AT %M87.1 : Bool;   // Znacznik sterowania w trybie sieć
   CB_CMD_P4 AT %M88.3 : Bool;   // Znacznik polecenia on/off przekaźnik napędu
   Set_HWork_P4 AT %M88.5 : Bool;   // Znacznik ustawienia aktywnej do pracy (po porównaniu liczników pracy)
   Is_extras_K1_P4 AT %M88.6 : Bool;   // Znacznik motor dodatkowy nr 1
   Set_50Hz_P4 AT %M89.0 : Bool;   // Znacznik pamięci podtrzymujący przełączenie na sieć
   setSUPV_FP4 AT %M89.3 : Bool;   // Znacznik polecenia startu z falownika
   IsRun_P4 AT %M89.4 : Bool;   // Potwierdzenie pracy
   setSUPV_SP4 AT %M89.5 : Bool;   // Znacznik polecenia startu z sieci
   Hour_Work_P4 AT %MD29 : DWord;   // Licznik pracy
   resetFault_SoftStart_P4 AT %M50.3 : Bool;   // sygnał resetu softstart
   bitH_Alarm_P4 AT %M28.0 : Bool;   // Alarm - kopia bitu z instancji statusu napędu
   bitH_rezerwa_P4 AT %M28.1 : Bool;   // rez
   bitH_REM_P4 AT %M28.2 : Bool;   // Zdalna - kopia bitu z instancji statusu napędu
   bitH_RUN_P4 AT %M28.3 : Bool;   // Praca - kopia bitu z instancji statusu napędu
   bitH_OFF_P4 AT %M28.4 : Bool;   // Polecenie OFF - kopia bitu z instancji statusu napędu
   bitH_ON_P4 AT %M28.5 : Bool;   // Polecenie ON - kopia bitu z instancji statusu napędu
   bitH_Res_P4 AT %M28.6 : Bool;   // Reset - kopia bitu z instancji statusu napędu
   bitH_Aut_Man_P4 AT %M28.7 : Bool;   // Aut=1 Man=0 - kopia bitu z instancji statusu napędu
   Is_extras_K3_P4 AT %M90.0 : Bool;   // Znacznik motor dodatkowy nr 3
   Is_extras_K2_P4 AT %M88.7 : Bool;   // Znacznik motor dodatkowy nr 2
   off_add_K1_P4 AT %M53.1 : Bool;   // sterowanie wyłączeniem selektywnym dodatkowej
   off_add_K2_P4 AT %M53.2 : Bool;   // sterowanie wyłączeniem selektywnym dodatkowej
   off_add_K3_P4 AT %M53.3 : Bool;   // sterowanie wyłączeniem selektywnym dodatkowej
   off_add_K4_P4 AT %M53.7 : Bool;   // sterowanie wyłączeniem selektywnym dodatkowej
   CMD_ErrorSet_NetworkP4 AT %M89.1 : Bool;   // Znacznik sterowania awaryjnego pracą pompy bez falownika
   Mem_Res_setCMD_MC_P4 AT %M89.2 : Bool;   // pamięć zbocza załączenia timera blokowania stycznika falowni P1
END_VAR

VAR_GLOBAL   // PLC tag table "PID"
   switc_manualPID AT %M206.5 : Bool;   // Przełacznik regulator PID na manualne zadawanie
   setUP_O2 AT %M300.3 : Bool;   // Znacznik generatora czasowego podnoszenia wartości zadanej ciśnienia
   setDown_O2 AT %M300.4 : Bool;   // Znacznik generatora czasowego obniżania wartości ciśnienia
END_VAR

VAR_GLOBAL   // PLC tag table "RTC"
   status_rd_sys_t AT %MW200 : Int;
   status_rd_loc_t AT %MW202 : Int;
   Ustaw_czas AT %M206.0 : Bool;
   trig_ustaw_czas AT %M206.1 : Bool;
   status_wr_sys_t AT %MW204 : Int;
   trig_pobierz_czas AT %M206.3 : Bool;
   Pobierz_czas AT %M206.2 : Bool;
END_VAR

VAR_GLOBAL   // PLC tag table "Sim"
   Sim_wiodaca AT %M1200.0 : Bool;
   Sim_SetUp_M25 AT %M1200.1 : Bool;
   Sim_SetDown_M25 AT %M1200.2 : Bool;
   Sim_aut_man AT %M1200.4 : Bool;
   Sim_SetDown_M27 AT %M1200.5 : Bool;
   simAnalogB5_Increm AT %M1041.0 : Bool;
   simAnalogB5_load AT %M1041.1 : Bool;
   simAnalogB5_Licznik AT %MW1042 : Word;
   simAnalogB5_decrem AT %M1041.4 : Bool;
   Tag_Start1 AT %M1041.2 : Bool;
   Tag_Start2 AT %M1041.3 : Bool;
   i AT %M1041.5 : Bool;
   Sim_daneMW AT %MD2000 : Real;
   "Ustaw alarm P3" AT %M1040.4 : Bool;
   STP_funkction_1 AT %M1041.7 : Bool;
   STP_funkction AT %M1041.6 : Bool;
   Sim_WarningHbar AT %M1200.3 : Bool;
END_VAR

VAR_GLOBAL   // PLC tag table "Sterowanie"
   INPUTstopAccident_Pompy AT %M84.3 : Bool;
   inputpowerOK_RS AT %M84.0 : Bool;
   "inputRem_P1-P4" AT %M84.1 : Bool;   // flaga tryb pracy zdalna / Tryb pracy 1=Auto, 0= Remontowe
   CMD_start_stop_inverter AT %M84.5 : Bool;   //    {ExternalWritable false}
   memRis_Foult_WiCC_PLC AT %M16.1 : Bool;   // Pamięć zbocza alarmu komunikacji WinCC-PLC
   memRis_WatchDog_HMI_PLC AT %M16.0 : Bool;   // Pamieć zbocza alarmu komunikacji KMI - PLC
   IsRem AT %M10.3 : Bool;   // Potwierdzenie trybu pracpomp 1=Auto, 0=Remontowe
   IsReady_Inverter AT %M10.7 : Bool;   // Znacznik gotowości falownika
   Mem_setMotor2 AT %M217.3 : Bool;   // Bit pamięci ustawienia pierwszego kompresora dodatkowego
   Mem_setMotor3 AT %M217.4 : Bool;   // Bit pamięci ustawienia drugiego kompresora dodatkowego
   mem_is_K1 AT %M218.1 : Bool;   // pamięć załaczenie znacznika pierwszej dodatkowego kompresora
   mem_Is_K2 AT %M218.2 : Bool;   // pamięć załaczenie znacznika pierwszej dodatkowego kompresora
   mem_Is_K3 AT %M218.3 : Bool;   // pamięć załaczenie znacznika wiodącego kompresora
   Is_extras_K1 AT %M219.2 : Bool;   // Znacznik dodatkowa 1
   Is_extras_K2 AT %M219.3 : Bool;   // Znacznik dodatkowa 2
   Is_up_Hz AT %M219.4 : Bool;   // Hz na wyjściu większe od minimalnych
   Mem_Res_setCMD_M9 AT %M11.7 : Bool;   // Pamięć zbocza blokowania stycznika falownik
   step_Hz_manual AT %MW26 : Int;   // Zmienna kroku ładowania Hz w trybie manual
   BarPress_Max AT %M219.6 : Bool;
   Set_50Hz AT %M219.7 : Bool;   // Znacznik pomocniczy dla procedury miękiego przełączenia Hz na falowniku
   mem_Triger_PowerOK AT %M220.0 : Bool;   // pamięć zbocza powroru zasilania
   Reset_HWork_errer AT %M220.1 : Bool;   // Kasowanie błędu ustawiania znaczników pracy od czasu
   Tmp_Set_SV AT %M220.4 : Bool;   // Znacznik ustawiania tymczasowej wartości Hz
   Rst_Driver_Max_presure AT %M221.6 : Bool;   // Znacznika awaryjnego wyłączenia od max ciśnienia napędu pracującego w trybie awaryjnym
   Switch_set_OverCurrentInverer AT %M10.0 : Bool;   // Przełącznik wyboru źródła zadawania wartości granicznej dopuszczalnego prądy falownika
   memZboczeN_wylK1 AT %M1101.0 : Bool;   // pamięć zbocza opadającego wyłaczenie dodatkowego 1
   srt50Hz_inverter_Level1 AT %M206.6 : Bool;   // Ustawienie 50 Hz w czasie wyłączenia dodatkowej Poziom 1
   isSetXXHz AT %M1101.1 : Bool;   // bit zatrzasku pamieci zboczaNeylK1
   RS_Zbocze_bar AT %M13.4 : Bool;   // Znacznik przekazujący info czy zbocze ciśnienieanarasta czy opada
   "inputready_Inverter_P1-P4" AT %M84.4 : Bool;   // gotowość faloenika
   Is_loading_K3 AT %M218.0 : Bool;   // Znacznik pompy wiodącej
   setPID_Pompy AT %M300.2 : Bool;   // Znacznik załączenie, regulacji falownika
   setMotor3 AT %M300.1 : Bool;   // Znacznik ustwienie dodatkowej dmuchawy nr2
   FC2_Set_50Hz AT %M15.0 : Bool;   // Zancznik ustalenia 50Hz
   Reset_Motor4_AlarmPresure AT %M90.2 : Bool;   // Znacznik wyłaczenia awaryjnego dmuchawy dodatkowej (alarm od ciśnienia)
   Reset_Motor4_AlarmOver AT %M90.3 : Bool;   // Znacznik wyłaczenia awaryjnego dmuchawy dodatkowej (alarm od przeciązenia)
   CMD_faultInverter AT %M90.4 : Bool;   // Znacznik awaria falownika
   CMD_faultP1 AT %M90.5 : Bool;   // Znacznik sygnalizacja awarii
   CMD_faultP2 AT %M90.6 : Bool;   // Znacznik sygnalizacja awarii
   CMD_faultP3 AT %M90.7 : Bool;   // Znacznik sygnalizacja awarii
   CMD_faultP4 AT %M91.0 : Bool;   // Znacznik sygnalizacja awarii
   setMotor4 AT %M300.6 : Bool;   // Znacznik ustwienie dodatkowej dmuchawy nr3
   memEdge_IsAut_pump AT %M19.1 : Bool;   // bit pamieci zbocza dla sygnału automatyczna praca pomp
   Mem_setMotor4 AT %M217.5 : Bool;   // Bit pamięci ustawienia trzeciej dodatkowej
   Is_extras_K3 AT %M221.7 : Bool;   // Znacznik dodatkowa 3
   memTrigSetAutomat AT %M19.2 : Bool;   // pamięć zbocza załaczenia trybu automat porzez stacyjki pomp
   memTrigManualFB1 AT %M19.7 : Bool;   // pamięć zbocza kontroli przełączników na HMI
   statMiasto AT %M54.0 : Bool;   // flaga start przetłaczanie - miasto
   statMagistrala AT %M54.1 : Bool;   // flaga start dosilanie - magistrala
   memTrigerStopAwariaPomp AT %M208.4 : Bool;   // pamięć zbocza dla zaczenia sygnalizacji wciśnięcia grzybka
   Reset_Motor3Alarm AT %M221.2 : Bool;   // Znacznik wyłączenia awaryjnego pompydodatkowej
   QW64 AT %QW64 : Int;   // Wartość Hz przekazywana na wyjście falownika
   inputrunInverter_ AT %M84.2 : Bool;   // Potwierdzenie załączeniea falownika
   Reset_Motor3_AlarmOver AT %M221.0 : Bool;   // Znacznik wyłaczenia awaryjnego pompy dodatkowej (alarm od ciśnienia)
   Reset_Motor3_AlarmPresure AT %M220.6 : Bool;   // Znacznik wyłaczenia awaryjnego pompydodatkowej (alarm od ciśnienia)
   IW166 AT %IW166 : Word;   // Sygnał z invertera aktualne Hz
   Static_1 AT %MD222 : Real;
   IsCurrentOverloadInverter AT %M11.4 : Bool;   // Znacznik przeciążenie falownika kompresorów
   Reset_Motor2_AlarmPresure AT %M220.5 : Bool;   // Znacznik wyłaczenia awaryjnego pompydodatkowej (alarm od ciśnienia)
   Reset_Motor2Alarm AT %M221.1 : Bool;   // Znacznik wyłączenia awaryjnego pompy dodatkowej
   IsRunInverter1 AT %M211.2 : Bool;   // Potwierdzenie pracy falownika kompresorów
   IsModeAut AT %M12.3 : Bool;   // Znacznik tryb automat dla
   IW164 AT %IW164 : Word;   // wejście analogowe   {ExternalWritable false}
   ActCurrent_Supply_Inverter AT %MD212 : DWord;   // Aktualny prąd obciążenia falownika
   Reset_Motor2_AlarmOver AT %M220.7 : Bool;   // Znacznik wyłaczenia awaryjnego pompydodatkowej (alarm od ciśnienia)
   setMotor2 AT %M300.0 : Bool;   // Znacznik ustwienie dodatkowej dmuchawy nr1 / Znacznik ustwienie dodatkowej pompy nr1
   zbocze_dod_zegar AT %M93.7 : Bool;
   Is_PowerRS5_OK AT %M11.3 : Bool;   // Zasilanie RS Zasuwy
   is_Aut_Z9 AT %M84.6 : Bool;   // bit stausu automat zasuwy Z9
   Reset_Motor4Alarm AT %M90.1 : Bool;   // Znacznik wyłączenie od alarmu dodatkowej 3   {ExternalVisible false}
   FB9_Set_Motor3 AT %M220.3 : Bool;   // Znacznik dodatkowej pompy dla funkcji FB8 I / Znacznik dodakowapompa 2 dla funkcji FB8 I
   FB9_Set_Motor2 AT %M220.2 : Bool;   // Znacznik dodatkowej pompy dla funkcji FB8 I / Znacznik dodakowapompa 1 dla funkcji FB8 I
   FB9_Set_Motor4 AT %M300.5 : Bool;   // Znacznik dodatkowej pompy dla funkcji FB8 I / Znacznik dodakowapompa 3 dla funkcji FB8 I
END_VAR

VAR_GLOBAL   // PLC tag table "Tag VLV01"
   Valve_Bit_K AT %M20.6 : Bool;   // Bit-6 kasowanie alarmu
   IN_STAT_Velv01 AT %MW20 : Word;   // Wejściowe słowo statusu napędu
   "Valve_Bit_A/R" AT %M20.7 : Bool;   // Bit trybu pracy napędu
   Valve_Bit_C AT %M20.5 : Bool;   // Rozkaz zamykania
   Valve_Bit_Open AT %M20.4 : Bool;   // Rozkaz otwieranie
   Valve_BIT_A AT %M20.0 : Bool;   // Bit gotowośći / awarii
   Byte_Wekt_Valve01 AT %MW24 : Word;   // Out- słowo wektora napędu
   "Bit_0-Wekt_Valve01" AT %M21.0 : Bool;   // Bit Alarm/Gotowość (Alarm-=1, gotowość=0)
   "Bit_1-Wekt_Valve01" AT %M21.1 : Bool;   // Bit potwierdzenia otwarcia
   "Bit_2-Wekt_Valve01" AT %M21.2 : Bool;   // Bit wyboru trybu Zdalne=1 Remontowe=0
   "Bit_3-Wek_Valve01" AT %M21.3 : Bool;   // Bit potwierdzenia zamknięcia
   "Bit_4-Wek_Valve01" AT %M21.4 : Bool;   // Bit rozkazu na otwieranie
   "Bit_5-Wekt-Valve01" AT %M21.5 : Bool;   // Bit rozkazu na zamykanie
   "Bit_6-Wekt-Valve01" AT %M21.6 : Bool;   // Bit kasowania
   "Bit_7-Wekt-Valve01" AT %M21.7 : Bool;   // Bit rodzaju sterowania aut =1 /manual= 0
   Byte_Wekt_Valve01_L AT %MB21 : Byte;   // Lewy byte wektora napędu
   Byte_Wekt_Valve01_R AT %MB20 : Byte;   // Prawy byte wektora napędu
   ByteH_Status_P1 AT %MB22 : Byte;   // status napędu
END_VAR

VAR_GLOBAL   // PLC tag table "Z11-Z12"
   inputREM_ZASUWY AT %M86.0 : Bool;
END_VAR

VAR_GLOBAL   // PLC tag table "Z11"
   isReadyZ11 AT %M85.3 : Bool;
   inputAwariaMomentZ11 AT %M85.4 : Bool;
   inputOtwartaZ11 AT %M85.5 : Bool;
   inputZamkniętaZ11 AT %M85.6 : Bool;
   inputRuchZ11 AT %M85.7 : Bool;
   setSVMO_Z11 AT %M13.6 : Bool;   // Znacznik polecenia otwórz w trybie automat
   inputmodeAutZ11 AT %M17.6 : Bool;   // Znacznik trybu pracy 1=Aut, 0=Rem
   inputAumalokalneZ11 AT %M87.2 : Bool;
   inputAumaautomatZ11 AT %M87.3 : Bool;
   inputAumagotowośćZ11 AT %M87.4 : Bool;
   inputAumaawariaZ11 AT %M87.5 : Bool;
   setSVMC_Z11 AT %M13.7 : Bool;   // Znacznik polecenia zamknij w trybie automat
   CMD_Open_Z11 AT %M33.3 : Bool;   // załącz otwieranie Z11
   CMD_Close_Z11 AT %M33.4 : Bool;   // załącz zamykanie Z11
   CMD_Awaria_Z11 AT %M91.2 : Bool;   // Awaria zbiorcza
   setAlarm_Moment_Z11 AT %M91.3 : Bool;   // znacznik alarmu od momentówki w trybie zdalnym (aut/mamnual)
   bitH_Alarm_Z11 AT %M95.0 : Bool;   // Alarm - kopia sygału z instancji DB10
   bitH_Open_Z11 AT %M95.1 : Bool;   // Otwarta - kopia sygału z instancji DB10
   bitH_REM_Z11 AT %M95.2 : Bool;   // Zdalne - kopia sygału z instancji DB10
   bitH_Close_Z11 AT %M95.3 : Bool;   // Zamknięta - kopia sygału z instancji DB10
   bitH_Opening_Z11 AT %M95.4 : Bool;   // sygnał otwórz- kopia sygału z instancji DB10
   bitH_Res_Z11 AT %M95.6 : Bool;   // sygnał reset - kopia sygału z instancji DB10
   bitH_Aut_Man_Z11 AT %M95.7 : Bool;   // sygnał aut=1, manual =0 - kopia sygału z instancji DB10
   bitH_Closing_Z11 AT %M95.5 : Bool;   // sygnał zamknij- kopia sygału z instancji DB10
   Byte_Status_Z11 AT %MB95 : Byte;   // status napędu
END_VAR

VAR_GLOBAL   // PLC tag table "Z12"
   isReadyZ12 AT %M86.5 : Bool;
   inputAwariaMomentZ12 AT %M86.1 : Bool;
   inputZamkniętaZ12 AT %M86.3 : Bool;
   imputRuchZ12 AT %M86.4 : Bool;
   setSVMO_Z12 AT %M86.6 : Bool;   // Znacznik polecenia otwórz w trybie automat
   inputmodeAutZ12 AT %M86.7 : Bool;   // Znacznik trybu pracy 1=Aut, 0=Rem
   inputAumalokalneZ12 AT %M87.6 : Bool;
   inputAumaautomatZ12 AT %M87.7 : Bool;
   inputAumagotowośćZ12 AT %M88.0 : Bool;
   inputAumaawariaZ12 AT %M88.1 : Bool;
   setSVMC_Z12 AT %M88.2 : Bool;   // Znacznik polecenia zamknij w trybie automat
   CMD_Open_Z12 AT %M33.5 : Bool;   // załącz otwieranie Z11
   CMD_Close_Z12 AT %M33.6 : Bool;   // załącz zamykanie Z11
   CMD_Awaria_Z12 AT %M91.1 : Bool;   // Awaria zbiorcza
   setAlarm_Moment_Z12 AT %M91.4 : Bool;   // znacznik alarmu od momentówki w trybie zdalnym (aut/mamnual)
   bitH_Alarm_Z12 AT %M97.0 : Bool;   // Alarm - kopia sygału z instancji DB10
   bitH_Open_Z12 AT %M97.1 : Bool;   // Otwarta - kopia sygału z instancji DB10
   bitH_REM_Z12 AT %M97.2 : Bool;   // Zdalne - kopia sygału z instancji DB10
   bitH_Close_Z12 AT %M97.3 : Bool;   // Zamknięta - kopia sygału z instancji DB10
   bitH_Opening_Z12 AT %M97.4 : Bool;   // sygnał otwórz- kopia sygału z instancji DB10
   bitH_Closing_Z12 AT %M97.5 : Bool;   // sygnał zamknij- kopia sygału z instancji DB10
   bitH_Res_Z12 AT %M97.6 : Bool;   // sygnał reset - kopia sygału z instancji DB10
   bitH_Aut_Man_Z12 AT %M97.7 : Bool;   // sygnał aut=1, manual =0 - kopia sygału z instancji DB10
   inputOtwartaZ12 AT %M86.2 : Bool;
   Byte_Status_Z12 AT %MB97 : Byte;   // status napędu
END_VAR

TYPE "stt_OB82"
// stored: IsFailsafeCompliant false
   STRUCT
      ErrorTimestamp : DTL;   // //time error occurs
      IO_State : Word;   // //Contains the I/O status of the diagnostics-capable module.
      LADDR : HW_ANY;   // //HW-ID
      Channel : UInt;   // //Channel number
      MultiError : Bool;   // //= 1, if there is more than one error
   END_STRUCT;
END_TYPE

TYPE "typVARIANT"
// stored: IsFailsafeCompliant false
   STRUCT
      VARIANT : Array[0..1] of Bool;
   END_STRUCT;
END_TYPE

TYPE "typeDataInverter_Byte"
// stored: IsFailsafeCompliant false
   STRUCT
      typeDataInverter_byte : Array[0..0] of Byte;   // Typ dane byte, falownik
   END_STRUCT;
END_TYPE

TYPE "typeDataInverter_DWord"
// stored: IsFailsafeCompliant false
   STRUCT
      typeDataInverter_Dword : Array[0..0] of DInt;   // dane dword, falownik
   END_STRUCT;
END_TYPE

TYPE "typeDataInverter_Real"
// stored: IsFailsafeCompliant false
   STRUCT
      typeDataInverter_real : Array[0..0] of Real;   // dane real, falownik
   END_STRUCT;
END_TYPE

TYPE "typeDataInverter_Word"
// stored: IsFailsafeCompliant false
   STRUCT
      typeDataInverter_int : Array[0..0] of Int;   // Typ danej Int, falownik
   END_STRUCT;
END_TYPE

TYPE "typeDataMPP04_Int"
// stored: IsFailsafeCompliant false
   STRUCT
      data : Array[0..1] of Int;
   END_STRUCT;
END_TYPE

TYPE "typeDataMPP04_int_1"
// stored: IsFailsafeCompliant false
   STRUCT
      data : Array[0..0] of Int;
   END_STRUCT;
END_TYPE

TYPE "typeDataMPP04_real"
// stored: IsFailsafeCompliant false
   STRUCT
      data : Array[0..0] of Real;
   END_STRUCT;
END_TYPE

TYPE "typeModbusCommLoad"
// stored: IsFailsafeCompliant false
   STRUCT
      done : Bool := FALSE;   // Boolean indicating completion without error
      error : Bool := FALSE;   // Boolean indicating completion with error
      status : Word := W#16#0;   // Status or error code of the completed operation
      errorStatus : Word := W#16#0;   // Error code of the faulty operation
   END_STRUCT;
END_TYPE

TYPE "typeModbusMaster"
// stored: IsFailsafeCompliant false
   STRUCT
      req : Bool := FALSE;   // The enable to initiate a Modbus master request
      mbAddr : UInt;   // The station address of the Modbus slave
      mode : USInt := 0;   // Specifies a read, write, or diagnostic operation
      dataAddr : UDInt := 0;   // The Modbus data address
      dataLen : UInt := 0;   // The Modbus data length
      done : Bool := FALSE;   // Boolean indicating completion without error
      busy : Bool := FALSE;   // Boolean indicating operation in progress
      error : Bool := FALSE;   // Boolean indicating completion with error
      status : Word := W#16#0;   // Status or error code of the completed operation
      errorStatus : Word := W#16#0;   // Error code of the faulty operation
   END_STRUCT;
END_TYPE

TYPE "typeModbusSlave"
// stored: IsFailsafeCompliant false
   STRUCT
      NDR : Bool := FALSE;   // New data ready: 1: Indicates that data has been read by the Modbus master No new data
      mbAddr : UInt;   // Station address of the Modbus slave (address range: 0 to 255)
      done : Bool := FALSE;   // Boolean indicating completion without error
      dr : Bool := FALSE;   // Read data: 0: No data read1: Indicates that data has been read by the Modbus master
      error : Bool := FALSE;   // Boolean indicating completion with error
      status : Word := W#16#0;   // Status or error code of the completed operation
      errorStatus : Word := W#16#0;   // Error code of the faulty operation
   END_STRUCT;
END_TYPE

DATA_BLOCK "db10organizacyjna"   // DB10
TITLE = Instance SCADA
{ S7_Optimized_Access := 'FALSE' }
AUTHOR : RTecmer
VERSION : 0.1
// stored: AutoNumber false, DBAccessibleFromOPCUA true, IsOnlyStoredInLoadMemory false, IsWriteProtectedInAS false
   VAR
      Clock : Time;
      Watchdog : Int;
      insPompa1 : Word;
      insPompa2 : Word;
      insPompa3 : Word;
      insPompa4 : Word;
      instB6_bar_act_miasto : Real;   // Ciśnienie B6 miasto [Real]
      instB5_bar_act_magistrala : Real;   // Ciśnienie B5 magistrala [Real]
      actPozycja_Z10 : Word;   // Aktualna pozycja Z10 [%]
      errorModbusRTU_SCADA : Word;   // awaria modbus rtu falownik bit 0, przepływomierz pompownia bit 1, przepływomierz magistra bit 2, sterownik MT101 bit 3
      HourCounterP1 : DWord;   // Counter Work
      HourCounterP2 : DWord;   // Counter Work
      HourCounterP3 : DWord;   // Counter Work
      HourCounterP4 : DWord;
      TimeHz : Int := 45;
      Time_ONK1 : Int := 110;
      Time_ONK2 : Int := 300;
      Time_OFFK1 : Int := 5;
      Time_OFFK2 : Int := 2;
      "PID_Compact_1_sPid_Cmpt.r_Sp_Hlm" : Real := 2.2;
      "PID_Compact_1_sPid_Cmpt.r_Sp_LIm" : Real := 1.5;
      set_Hz_P1P4 : Real;   // Aktualne Hz na falowniku
      setpoint_SV_bar : Real := 1.8;   // Zadana wartość ciśnienie do PID [bar]
      set_min_press_bar_B8 : Real := 0.0;   // minimalne ciśnienie bezpieczeństwa [bar] B8
      instFlowDN225_act_Q1 : Real;   // aktualny przepływ Q1 pompownia
      reset_modbus_TCP : Bool;   // reset komunikacji modbus TCP
      instB7_bar_act_pompownia : Real := 0.28;   // aktualne
      min_Bar_set : Real := 1.7;   // Minimalne ciśnienie zadane
      max_Bar_set : Real := 2.7;   // Maxymalne ciśnienie zadane
      actTime : Real;   // aktualny czas
      "pos_Setpint_SV bar" : Real;   // Aktualna wartość zadanaego ciśnienie
      act_stanP1 : Int;   // Zmienna na potzrzeby trenów pracy pompy
      act_statnP2 : Int;   // Zmienna na potzrzeby trenów pracy pompy
      act_stanP3 : Int;   // Zmienna na potzrzeby trenów pracy pompy
      act_stanP4 : Int;
      instSumFlowDN225_Q1 : Real;   // Aktualny przepływ na wlocie oczyszczalni m3/h
      switch_ModelSterowania : Word := 1;   // Zmienna przyjmująca wartość dziesiętnią oznaczającą model sterowania
      instB8_bar_act_suchobieg : Real;   // Ciśnienie suchobiegu (0-1bar)
      "alarms only" : Word;   // Instancja alarmów (bit 146.4 - Error Modbus),(bit 146.5-Warning Modbau)
      inverterPomp_Status : Word;   // Status falownika pomp
      inst_act_Current_Inverters : Real;   // Aktualny prąd falownika [A]
      set_press_bar_Max : Real := 7.888;   // Maxymalne dopuszczalne ciśnienie w rurociągu [bar]
      ampere_Max : Real := 56.0;   // Edytowalne - Maxymalne dopuszczalne przeciążenie [A]
      act_Hz_Inverter_1 : Real;   // Aktualne Hz na falowniku
      ins_ModeWorkContactronP1 : Word;   // Zmienna przechowująca informację o stanie napędu (0-postój, 1-falownik, 2-sieć)
      ins_ModeWorkContactronP2 : Word;   // Zmienna przechowująca informację o stanie napędu (0-postój, 1-falownik, 2-sieć)
      ins_ModeWorkContactronP3 : Word;   // Zmienna przechowująca informację o stanie napędu (0-postój, 1-falownik, 2-sieć)
      ins_ModeWorkContactronP4 : Word;   // Zmienna przechowująca informację o stanie napędu (0-postój, 1-falownik, 2-sieć)
      instB9_bar_act_Granica : Real;   // Wartość bar w sterowanym zbiorniku
      PV_HWrn_set_correct : Real := 2.1;   // Wspóczninik służący wprowadzeniu korekty ostrzeżenia przekroczenia wartości zadanej bar
      PV_LWrn_set_correct : Real := 0.6;   // Wspóczninik służący wprowadzeniu korekty ostrzeżenia zbyt niskia wartości bar w stosunku do zadanej
      TimeHistere_set_bar : Int := 1;   // Czas zwłoki przed zmianą bar zadanego podczas redukcji azotu
      avg_bar : Real;   // srednia wartość ciśnienie
      RTU_Fal_1errorStatus : Word;   // Status błędu komunikacji Modbus RTU
      RTU_MPP04_1errorStatus : Word;   // Status błędu komunikacji Modbus RTU
      RTU_MPP04_2errorStatus : Word;   // Status błędu komunikacji Modbus RTU
      RTU_MT101 : Word;   // Status błędu komunikacji Modbus RTU
      RTU_stepRESET : Bool := 1;   // Krok pętli Modbus RTU na potrzeby SCADA (RESET)
      setRTU_Error : Bool;   // Znacznik błedu modbus RTU
      instSecStart_City_1 : Int;   // Sekundy start przetłaczanie
      instSecStop_City_1 : Int;   // Sekundy stop przetłaczanie
      instSecStart_Replen_1 : Int;   // Sekundy start dosilanie
      instSecStop_Replen_1 : Int;   // Sekundy stop dosilanie
      CounterOverTempFa : Int;   // Licznik wystąpienia usterki przegrzania
      instSecStart_Filling_1 : Int;   // Sekundy start napełniania
      instSecStop_Filling_1 : Int;   // Sekundy stop napełniania
      CounterOverVoltFal : Int;   // Licznik wystapienia usterki wysokie VDC
      instHourStart_Filling_1 : Int;   // Godzina start napełniania
      instMinutStart_Filling : Int;   // Minuta start napełniania
      instHourStop_Filling_1 : Int;   // Godzina stop napełniania
      instMinutStopt_Filling : Int;   // Minuta stop napełniania
      instFlowDN500_act_Q2 : Real;   // Aktualna wartośc przepływu Q2 magistrala
      instSumFlowDN500_Q2 : Real;   // Aktualna wartośc sumy przepywu Q2 magistrala
      instHourStart_Filling : DTL;   // Godzina start napełniania
      instHourStop_Filling : DTL;   // Godzina stop napełniania
      instHourStart_City : DTL;   // Godzina start przetłaczanie miasto DN225
      instHourStop_City : DTL;   // Godzina stop przetłaczanie miasto DN225
      instHourStart_Replen : DTL;   // Godzina start dosilanie DN500
      instHourStop_Replen : DTL;   // Godzina stop dosilanie DN500
      actQ1_przepyw_pompownia_Int : Word;   // Aktualny przepływ na Q1 pompownia
      actQ2_przepyw_pompownia_Int : Word;   // Aktualny przepływ na Q2 pompownia
      inst_sum_FlowDN255_act_Q2_int : Word;   // aktualna suma przepływu Q1 (int)
      inst_sumFlowDN500_act_Q2_int : Word;   // aktualna suma przepływu Q2 (int)
      instHourStart_City_1 : Int;   // Godzina start przetłaczanie miasto DN225
      instMinutStart_City : Int;   // Minuty start przetłaczanie miasto DN225
      instHourStop_City_1 : Int;   // Godzina stop przetłaczanie miasto DN225
      instMinutStopt_City : Int;   // Minuty stop przetłaczanie miasto DN225
      instHourStart_Replen_1 : Int;   // Godzina start dosilanie magistrala DN500
      instMinutStart_Replen : Int;   // Minuty start dosilanie magistrala DN500
      instHourStop_Replen_1 : Int;   // Godzina stop dosilanie magistrala DN500
      instMinutStopt_Replen : Int;   // Minuty stop dosilanie magistrala DN500
      instvValveZ1 : Word;   // Zasuwa zbiornik - spust zbiornik 1
      instvValveZ2 : Word;   // Zasuwa zbiornik - zasilanie zbiornik 1
      instvValveZ3 : Word;   // Zasuwa zbiornik - spust zbiornik 2
      instvValveZ4 : Word;   // Zasuwa zbiornik - zasilanie zbiornik 2
      instvValveZ5 : Word;   // Zasuwa zbiornik - spust zbiornik 3
      instvValveZ6 : Word;   // Zasuwa zbiornik - zasilanie zbiornik 3
      instvValveZ7 : Word;   // Zasuwa zbiornik - spust zbiornik 4
      instvValveZ8 : Word;   // Zasuwa zbiornik - zasilanie zbiornik 4
      instvValveZ9 : Word;   // Zasuwa suchobieg
      instvValveZ10 : Word;   // Zasuwa zbiornik regulowana - zasilanie
      actHour : Int;   // Godzina start dosilanie magistrala DN500
      actMinut : Int;   // aktualny czas
      actSec : Int := 0;   // aktualny czas
   END_VAR
BEGIN
END_DATA_BLOCK

DATA_BLOCK "dbHoldRegSlave_to_MT101"   // DB100
{ S7_Optimized_Access := 'FALSE' }
VERSION : 0.1
// stored: AutoNumber false, DBAccessibleFromOPCUA true, IsOnlyStoredInLoadMemory false, IsWriteProtectedInAS false
   VAR
      instPump1 : Word := 33924;   // 40001 Pompa Status M1
      instPump2 : Word := 33924;   // 40002 Pompa Status M2
      instPump3 : Word := 33924;   // 40003 Pompa Status M3
      instPump4 : Word := 33924;   // 40004 Pompa Status M4
      instvValveZ1 : Word := 33924;   // 40005 Zasuwa Status Z1
      instvValveZ2 : Word := 33924;   // 40006 Zasuwa Status Z2
      instvValveZ3 : Word := 33924;   // 40007 Zasuwa Status Z3
      instvValveZ4 : Word := 33924;   // 40008 Zasuwa Status Z4
      instvValveZ5 : Word := 33924;   // 40009 Zasuwa Status Z5
      instvValveZ6 : Word := 33924;   // 40010 Zasuwa Status Z6
      instvValveZ7 : Word := 33924;   // 40011 Zasuwa Status Z7
      instvValveZ8 : Word := 33924;   // 40012 Zasuwa Status Z8
      instvValveZ9 : Word := 33924;   // 40013 Zasuwa Status Z9
      instvValveZ10 : Word := 33924;   // 40014 Zasuwa Status Z10
      instvValveZ11 : Word := 33924;   // 40015 Zasuwa Status Z11
      instvValveZ12 : Word := 33924;   // 40016 Zasuwa Status Z12
      instControllDrivers_1 : Int := 0;   // Bity sterowania napędami (start, stop, otwórz, zamknij) / 40017 Bity sterowania napędami (start, stop, otwórz, zamknij) Pompami M1-M4, Zasuwami Z1, Z2, Z3, Z4
      instControllDrivers_2 : Int := 0;   // Bity przełączenia trybu pracy napędów / 40018 Bity sterowania napędami ( otwórz, zamknij, start, stop) Zasuwami Z5, Z6, Z7, Z8, Z9, Z10, Z11, Z12
      instConrol_ManAut_1 : Int := 0;   // Bity przełączenia trybu pracy napędów / 40019 Bity przełączenia trybu pracy napędów M1-M4, Zasuwami Z1, Z2, Z3, Z4
      instConrol_ManAut_2 : Int := 0;   // Bity przełączenia trybu pracy napędów / 40020 Bity przełączenia trybu pracy napędów Z5, Z6, Z7, Z8, Z9, Z10, Z11, Z12
      instLevelTank1 : Int := 0;   // Poziom zbiornik / 40021 Poziom zbiornik
      instLevelTank2 : Int := 0;   // Poziom zbiornik / 40022 Poziom zbiornik
      instLevelTank3 : Int := 0;   // Poziom zbiornik / 40023 Poziom zbiornik
      instLevelTank4 : Int := 0;   // Poziom zbiornik / 40024 Poziom zbiornik
      instPosition_Z10 : Int;   // rezerwa / 40025 Zadawanie położenia Z10
      instClearFault1 : Int := 0;   // Bity kasowania alarmów napędów M1-M4, Z1 - Z12 / 40026 Bity kasowania alarmów napędów M1-M4, Z1 - Z12
      instSygSter_1 : Int := 2;   // rezerwa / 40027 Sygnały sterowania strategią pompownia - 0= wyłaczone, 1=dosilanie, 2=przetłaczanie,3=automat, 4=ręczne
      instSygSter_2 : Int := 1;   // 40028 Sygnały sterowania cyklem zbiorniki 0-wyłączone, 1=dobowy, 2=tygodniowy, 3=ręczne
      instCurrent_Inverter : Int := 0;   // 40029 Aktualny prądu falownika
      instHz_Inverter : Int := 0;   // 40030 Aktualne Hz na falowniku
      instLevelSetFilling : Real := 550.0;   // 40031 Zadany poziom napełniania
      instLevelSetEmptying : Real := 30.0;   // 40033 Zadany poziom opróżniania
      instSetbarDN225_B6 : Real := 6.6;   // 40035 Zadany ciśnienie tłóczenia kierunek miasto, Modbus 40035
      instSetbarDN500_B5 : Real := 7.0;   // 40037 Zadana ciśnienie dosilania kierunek dosilanie "0" Modbus 40037
      instSetBarMinB9 : Real := 6.5;   // 40039 Zadawana dolna granica ciśnienia studnia "Granica" Modbus 40039
      instB5bar_act : Real;   // 40041 Aktualne ciśnienie zasilania z sieci
      instB6bar_act : Real;   // 40043 Aktualne ciśnienie DN225 tłoczny
      instB7bar_act : Real;   // 40045 Aktualne ciśnienie DN225 pompy
      instB8bar_act : Real;   // 40047 Aktualne ciśnienie ssoncy pomp (zab. Suchobieg)
      instPozitionZ10_act : Real;   // 40049 Aktualna pozycja zasuwy Z10
      instFlowDN225_act : Real;   // 40051 Przepływ DN225 aktualny MIASTO
      instFlowDN225_sum : Real;   // 40053 SUMA przepływu Dolna DN225
      instFlowDN500_act : Real;   // 40055 Przepływ DN500 (l/s) aktualny, zasilanie zbiorników, DOSILANIE, Modbus 40055
      instFlowDN500_sum : Real;   // 40057 SUMA przepływu Dolna DN500 Modbus 40057
      instHourStart_Filling : Int := 0;   // 40059 Godzina start napełniania
      instMinutStart_Filling : Int := 5;   // 40060 Minuta start napełniania
      instHourStop_Filling : Int := 17;   // 40061 Godzina stop napełniania
      instMinutStopt_Filling : Int := 0;   // 40062 Minuta stop napełniania
      instHourStart_City : Int := 18;   // 40063 Godzina start przetłaczanie miasto DN225
      instMinutStart_City : Int := 0;   // 40064 Minuty start przetłaczanie miasto DN225
      instHourStop_City : Int := 23;   // 40065 Godzina stop przetłaczanie miasto DN225
      instMinutStopt_City : Int := 59;   // 40066 Minuty stop przetłaczanie miasto DN225
      instHourStart_Replen : Int := 18;   // 40067 Godzina start przetłaczanie magistrala DN500
      instMinutStart_Replen : Int := 0;   // 40068 Minuty start przetłaczanie magistrala DN500
      instHourStop_Replen : Int := 23;   // 40069 Godzina stop przetłaczanie magistrala DN500
      instMinutStopt_Replen : Int := 59;   // 40070 Minuty stop przetłaczanie magistrala DN500
   END_VAR
BEGIN
END_DATA_BLOCK

DATA_BLOCK "dbzarządzanie"   // DB91
TITLE = instacja zarz adzająca
{ S7_Optimized_Access := 'FALSE' }
AUTHOR : rtecmer
VERSION : 0.1
// blok danych pośrednicząc  pomiędzy warstwami
// stored: AutoNumber true, DBAccessibleFromOPCUA true, IsOnlyStoredInLoadMemory false, IsWriteProtectedInAS false
   VAR
      reset : Struct
         resetLicznikPracy_P1 : Bool;   // kasawanie licznika pracy
         resetLicznikPracy_P2 : Bool;   // kasawanie licznika pracy
         resetLicznikPracy_P3 : Bool;   // kasawanie licznika pracy
         resetLicznikPracy_P4 : Bool;   // kasawanie licznika pracy
      END_STRUCT;
      sterowanie_1 : Struct
         stop_falownik : Bool;   // zatrzymanie sterowania falownikiem
         tryb_automat : Bool;   // bit sygnalizacji pracy w automacie zestawu
         "alarm-warning" : Bool;   // alarm ostrzerzenie
         "alarm-modbus" : Bool;   // alarm modbus
         alarm_comunication_WinCC : Bool;   // alarm kominikacji wincc
         "alarm-comunication_HMI" : Bool;
         awaria_modbus_falownik : Bool;   // na potrzeby indentyfikacji awarii do tabeli alarów
         awaria_modbus_przepływ_pomp : Bool;   // na potrzeby indentyfikacji awarii do tabeli alarów
         awaria_modbus_przepływ_magist : Bool;   // na potrzeby indentyfikacji awarii do tabeli alarów
         awaria_modbus_mt101 : Bool;   // na potrzeby indentyfikacji awarii do tabeli alarów
         aktywna_P1 : Bool;
         aktywna_P2 : Bool;
         aktywna_P3 : Bool;
         aktywna_P4 : Bool;
         aktywna_Z11 : Bool;
         aktywna_Z12 : Bool;
         tempStrategia_pompownia : Int;   // Słowo tymczasowe przechwycone podczas wystapienia awarii niskiego ciśnienia magistrala
      END_STRUCT;
      awaria_falownika_F1 : Bool;   // Gotowość falownika 1
      awaria_falownika_F2 : Bool;   // Gotowość falownika 2
      brak_zasilania_RS : Bool;   // Brak zasilania
      instHourStart_Filling : Real;   // Godzina start napełniania
      instHourStop_Filling : Real;   // Godzina stop napełniania
      instHourStart_City : Real;   // Godzina start przetłaczanie miasto DN225
      instHourStop_City : Real;   // Godzina stop przetłaczanie miasto DN225
      instHourStart_Replen : Real;   // Godzina start dosilanie DN500
      instHourStop_Replen : Real;   // Godzina stop dosilanie DN500
      "Alarm analogs to HMI" : Struct   // Alarmy analogowe dla HMI
         "B5 Magistrala max" : Real := 8.5;   // alarm max
         "B6 Miasto max" : Real := 8.0;   // alarm max
         "B7 Pompownia max" : Real := 8.0;   // alarm max
         "B8 suchonieg min" : Real := 0.5;   // alarm min
         "Zbiornik max Nr_1" : Real := 558.0;   // alarm max
         "Zbiornik max Nr_2" : Real := 558.0;   // alarm max
         "Zbiornik max Nr_3" : Real := 558.0;   // alarm max
         "Zbiornik max Nr_4" : Real := 558.0;   // alarm max
      END_STRUCT;
   END_VAR
BEGIN
END_DATA_BLOCK

DATA_BLOCK "DB 333"   // DB333
{ S7_Optimized_Access := 'FALSE' }
AUTHOR : AWP_S7P
FAMILY : WEB
VERSION : 1.0
// stored: AutoNumber false, DBAccessibleFromOPCUA true, IsOnlyStoredInLoadMemory false, IsWriteProtectedInAS false
   VAR
      magic { ExternalAccessible := 'False'; ExternalVisible := 'False'; ExternalWritable := 'False'} : DWord := DW#16#41575043;
      consistency_tag { ExternalAccessible := 'False'; ExternalVisible := 'False'; ExternalWritable := 'False'} : DWord := DW#16#3B3640B8;
      db_version { ExternalAccessible := 'False'; ExternalVisible := 'False'; ExternalWritable := 'False'} : Word := W#16#0001;
      length { ExternalAccessible := 'False'; ExternalVisible := 'False'; ExternalWritable := 'False'} : UInt := 182;
      pagetab_of { ExternalAccessible := 'False'; ExternalVisible := 'False'; ExternalWritable := 'False'} : UInt := 92;
      pagetab_count { ExternalAccessible := 'False'; ExternalVisible := 'False'; ExternalWritable := 'False'} : UInt := 1;
      excludetab_of { ExternalAccessible := 'False'; ExternalVisible := 'False'; ExternalWritable := 'False'} : UInt := 102;
      excludetab_count { ExternalAccessible := 'False'; ExternalVisible := 'False'; ExternalWritable := 'False'} : UInt := 0;
      fragmentlist_of { ExternalAccessible := 'False'; ExternalVisible := 'False'; ExternalWritable := 'False'} : UInt := 102;
      fragmentlist_count { ExternalAccessible := 'False'; ExternalVisible := 'False'; ExternalWritable := 'False'} : UInt := 1;
      fragmenttab_of { ExternalAccessible := 'False'; ExternalVisible := 'False'; ExternalWritable := 'False'} : UInt := 110;
      fragmenttab_count { ExternalAccessible := 'False'; ExternalVisible := 'False'; ExternalWritable := 'False'} : UInt := 1;
      datatab_of { ExternalAccessible := 'False'; ExternalVisible := 'False'; ExternalWritable := 'False'} : UInt := 124;
      datatab_count { ExternalAccessible := 'False'; ExternalVisible := 'False'; ExternalWritable := 'False'} : UInt := 0;
      usenametab_of { ExternalAccessible := 'False'; ExternalVisible := 'False'; ExternalWritable := 'False'} : UInt := 124;
      usenametab_count { ExternalAccessible := 'False'; ExternalVisible := 'False'; ExternalWritable := 'False'} : UInt := 0;
      enumreftab_of { ExternalAccessible := 'False'; ExternalVisible := 'False'; ExternalWritable := 'False'} : UInt := 124;
      enumreftab_count { ExternalAccessible := 'False'; ExternalVisible := 'False'; ExternalWritable := 'False'} : UInt := 0;
      enumtab_of { ExternalAccessible := 'False'; ExternalVisible := 'False'; ExternalWritable := 'False'} : UInt := 124;
      enumtab_count { ExternalAccessible := 'False'; ExternalVisible := 'False'; ExternalWritable := 'False'} : UInt := 0;
      textlist_of { ExternalAccessible := 'False'; ExternalVisible := 'False'; ExternalWritable := 'False'} : UInt := 124;
      textlist_count { ExternalAccessible := 'False'; ExternalVisible := 'False'; ExternalWritable := 'False'} : UInt := 58;
      language_frag_tab_of { ExternalAccessible := 'False'; ExternalVisible := 'False'; ExternalWritable := 'False'} : UInt := 104;
      language_frag_tab_count { ExternalAccessible := 'False'; ExternalVisible := 'False'; ExternalWritable := 'False'} : UInt := 6;
      application_name { ExternalAccessible := 'False'; ExternalVisible := 'False'; ExternalWritable := 'False'} : UInt := 1;
      application_url { ExternalAccessible := 'False'; ExternalVisible := 'False'; ExternalWritable := 'False'} : UInt := 10;
      application_desc { ExternalAccessible := 'False'; ExternalVisible := 'False'; ExternalWritable := 'False'} : UInt := 20;
      enum_defs_fragment_start { ExternalAccessible := 'False'; ExternalVisible := 'False'; ExternalWritable := 'False'} : UInt := 0;
      enum_defs_fragment_count { ExternalAccessible := 'False'; ExternalVisible := 'False'; ExternalWritable := 'False'} : UInt := 0;
      commandstate { ExternalAccessible := 'False'; ExternalVisible := 'False'; ExternalWritable := 'False'} : Struct
         last_error { ExternalAccessible := 'False'; ExternalVisible := 'False'; ExternalWritable := 'False'} : Int := 0;
         debug_mode { ExternalAccessible := 'False'; ExternalVisible := 'False'; ExternalWritable := 'False'} : Int := 0;
         init { ExternalAccessible := 'False'; ExternalVisible := 'False'; ExternalWritable := 'False'} : Bool := True;
         deactivate { ExternalAccessible := 'False'; ExternalVisible := 'False'; ExternalWritable := 'False'} : Bool := False;
         initializing { ExternalAccessible := 'False'; ExternalVisible := 'False'; ExternalWritable := 'False'} : Bool := False;
         error { ExternalAccessible := 'False'; ExternalVisible := 'False'; ExternalWritable := 'False'} : Bool := False;
         deactivating { ExternalAccessible := 'False'; ExternalVisible := 'False'; ExternalWritable := 'False'} : Bool := False;
         deactivated { ExternalAccessible := 'False'; ExternalVisible := 'False'; ExternalWritable := 'False'} : Bool := False;
         initialized { ExternalAccessible := 'False'; ExternalVisible := 'False'; ExternalWritable := 'False'} : Bool := False;
         reserved1 { ExternalAccessible := 'False'; ExternalVisible := 'False'; ExternalWritable := 'False'} : Bool := False;
         reserved2 { ExternalAccessible := 'False'; ExternalVisible := 'False'; ExternalWritable := 'False'} : Byte := B#16#00;
      END_STRUCT;
      requesttab { ExternalAccessible := 'False'; ExternalVisible := 'False'; ExternalWritable := 'False'} : Array[1..4] of Struct
         page_index { ExternalAccessible := 'False'; ExternalVisible := 'False'; ExternalWritable := 'False'} : UInt;
         fragment_index { ExternalAccessible := 'False'; ExternalVisible := 'False'; ExternalWritable := 'False'} : UInt;
         continue { ExternalAccessible := 'False'; ExternalVisible := 'False'; ExternalWritable := 'False'} : Bool;
         "repeat" { ExternalAccessible := 'False'; ExternalVisible := 'False'; ExternalWritable := 'False'} : Bool;
         abort { ExternalAccessible := 'False'; ExternalVisible := 'False'; ExternalWritable := 'False'} : Bool;
         finish { ExternalAccessible := 'False'; ExternalVisible := 'False'; ExternalWritable := 'False'} : Bool;
         idle { ExternalAccessible := 'False'; ExternalVisible := 'False'; ExternalWritable := 'False'} : Bool;
         waiting { ExternalAccessible := 'False'; ExternalVisible := 'False'; ExternalWritable := 'False'} : Bool;
         sending { ExternalAccessible := 'False'; ExternalVisible := 'False'; ExternalWritable := 'False'} : Bool;
         aborting { ExternalAccessible := 'False'; ExternalVisible := 'False'; ExternalWritable := 'False'} : Bool;
         reserved3 { ExternalAccessible := 'False'; ExternalVisible := 'False'; ExternalWritable := 'False'} : Byte;
      END_STRUCT;
      pagetab { ExternalAccessible := 'False'; ExternalVisible := 'False'; ExternalWritable := 'False'} : Array[1..1] of Struct
         index { ExternalAccessible := 'False'; ExternalVisible := 'False'; ExternalWritable := 'False'} : UInt;
         url { ExternalAccessible := 'False'; ExternalVisible := 'False'; ExternalWritable := 'False'} : UInt;
         mime_type { ExternalAccessible := 'False'; ExternalVisible := 'False'; ExternalWritable := 'False'} : UInt;
         fragment_start { ExternalAccessible := 'False'; ExternalVisible := 'False'; ExternalWritable := 'False'} : UInt;
         fragment_num { ExternalAccessible := 'False'; ExternalVisible := 'False'; ExternalWritable := 'False'} : UInt;
      END_STRUCT;
      fragmentlist { ExternalAccessible := 'False'; ExternalVisible := 'False'; ExternalWritable := 'False'} : Array[1..1] of UInt;
      language_frag_tab { ExternalAccessible := 'False'; ExternalVisible := 'False'; ExternalWritable := 'False'} : Struct
         max_language { ExternalAccessible := 'False'; ExternalVisible := 'False'; ExternalWritable := 'False'} : UInt := 0;
         fragment_count { ExternalAccessible := 'False'; ExternalVisible := 'False'; ExternalWritable := 'False'} : UInt := 0;
         nolang_offset { ExternalAccessible := 'False'; ExternalVisible := 'False'; ExternalWritable := 'False'} : UInt := 0;
      END_STRUCT;
      fragmenttab { ExternalAccessible := 'False'; ExternalVisible := 'False'; ExternalWritable := 'False'} : Array[1..1] of Struct
         fragment_name { ExternalAccessible := 'False'; ExternalVisible := 'False'; ExternalWritable := 'False'} : UInt;
         fragment_type { ExternalAccessible := 'False'; ExternalVisible := 'False'; ExternalWritable := 'False'} : Byte;
         fragment_version { ExternalAccessible := 'False'; ExternalVisible := 'False'; ExternalWritable := 'False'} : Byte;
         content_db { ExternalAccessible := 'False'; ExternalVisible := 'False'; ExternalWritable := 'False'} : UInt;
         content_of { ExternalAccessible := 'False'; ExternalVisible := 'False'; ExternalWritable := 'False'} : UInt;
         content_length { ExternalAccessible := 'False'; ExternalVisible := 'False'; ExternalWritable := 'False'} : UInt;
         data_start { ExternalAccessible := 'False'; ExternalVisible := 'False'; ExternalWritable := 'False'} : UInt;
         data_num { ExternalAccessible := 'False'; ExternalVisible := 'False'; ExternalWritable := 'False'} : UInt;
      END_STRUCT;
      textlist { ExternalAccessible := 'False'; ExternalVisible := 'False'; ExternalWritable := 'False'} : Array[1..58] of Byte := 777777446F6C6E6100696E6465782E68746D00777777446F6C6E6100696E6465782E68746D00746578742F68746D6C00696E6465782E68746D00;
   END_VAR
BEGIN
   requesttab[1..4].page_index := 0;
   requesttab[1..4].fragment_index := 0;
   requesttab[1..4].continue := False;
   requesttab[1..4]."repeat" := False;
   requesttab[1..4].abort := False;
   requesttab[1..4].finish := False;
   requesttab[1..4].idle := False;
   requesttab[1..4].waiting := False;
   requesttab[1..4].sending := False;
   requesttab[1..4].aborting := False;
   requesttab[1..4].reserved3 := B#16#00;
   pagetab[1].index := 1;
   pagetab[1].url := 29;
   pagetab[1].mime_type := 39;
   pagetab[1].fragment_start := 1;
   pagetab[1].fragment_num := 1;
   fragmentlist[1] := 1;
   fragmenttab[1].fragment_name := 49;
   fragmenttab[1].fragment_type := B#16#00;
   fragmenttab[1].fragment_version := B#16#00;
   fragmenttab[1].content_db := 334;
   fragmenttab[1].content_of := 0;
   fragmenttab[1].content_length := 0;
   fragmenttab[1].data_start := 0;
   fragmenttab[1].data_num := 0;
END_DATA_BLOCK

DATA_BLOCK "DB 334"   // DB334
{ S7_Optimized_Access := 'FALSE' }
AUTHOR : AWP_S7P
FAMILY : WEB
VERSION : 0.1
// stored: AutoNumber false, DBAccessibleFromOPCUA true, IsOnlyStoredInLoadMemory true, IsWriteProtectedInAS false
   VAR
      MAGIC { ExternalAccessible := 'False'; ExternalVisible := 'False'; ExternalWritable := 'False'} : DWord := DW#16#4157_5046;
      CONSISTENCY_TAG { ExternalAccessible := 'False'; ExternalVisible := 'False'; ExternalWritable := 'False'} : DWord := 993411256;
   END_VAR
BEGIN
END_DATA_BLOCK

DATA_BLOCK "EX012_ErrorBuffer_OB82"   // DB103
TITLE = BufferOB82
{ S7_Optimized_Access := 'TRUE' }
AUTHOR : Gilewski
VERSION : 0.1
// Data block for OB82 buffer
// stored: AutoNumber false, DBAccessibleFromOPCUA true, IsOnlyStoredInLoadMemory false, IsRetainMemResEnabled false, IsWriteProtectedInAS false, MemoryReserve 100
   VAR RETAIN
      OB82ErrorCounter : USInt;   // //Counter for error buffer
      CounterDiagStatusUpdate : USInt;   // //Counter for another error
      ErrorDataOB82 { S7_SetPoint := 'True'} : Array[1..200] of "stt_OB82";   // //buffer for error from OB82
   END_VAR
BEGIN
END_DATA_BLOCK

DATA_BLOCK "DB31_HMI_AreaPointer"   // DB31
{ S7_Optimized_Access := 'FALSE' }
VERSION : 0.1
// stored: AutoNumber false, DBAccessibleFromOPCUA true, IsOnlyStoredInLoadMemory false, IsWriteProtectedInAS false
   VAR
      Coordination : Word;
      DateTime : DTL;
      JobMailbox : Array[0..3] of Word;
      DataRecord : Array[0..4] of Word;
      ProjectID : Word;
      ScreenNumber : Array[0..4] of Word;
      DateTimePLC : Struct
         DateTime : DTL;
         Reserve_01 : Word;
         Reserve_02 : Word;
      END_STRUCT;
      getPLCMode : Int;
      retValueTime : Word;
      cpuSatus : Bool;
   END_VAR
BEGIN
END_DATA_BLOCK

DATA_BLOCK "Dane_ComunicationControlHMI"   // DB29
TITLE = WatchDog HMI-Krata - S7-Krata
{ S7_Optimized_Access := 'FALSE' }
AUTHOR : rtecmer
VERSION : 0.1
// stored: AutoNumber true, DBAccessibleFromOPCUA true, IsOnlyStoredInLoadMemory false, IsWriteProtectedInAS false
   VAR
      Data_czas_loc : DTL;   // Zegar dla panelu HMI Krata
      WatchDog_WinCC : Word;   // Zmienna kordynująca kontrolę komunikacji od strony PC WinCC.
      SetFaultComunikation_Zasuwy : Int;   // Kontrola komunikacji z HMI
      Data_czas_sys : DTL;   // Zegar dla panelu HMI Krata
      Data_czasHMI : DTL;   // Zegar czytany z funkcji RTC (FC44) zapas
      tempCoordinationHMIRS5 : Int;   // Kontrola CoorditionHMI KDN
      tempWatchDog_WinCC : Word;   // Zmienna kordynująca kontrolę komunikacji od strony PC WinCC.
   END_VAR
BEGIN
END_DATA_BLOCK

DATA_BLOCK "Data_Czas_synch"   // DB32
{ S7_Optimized_Access := 'FALSE' }
VERSION : 0.1
// stored: AutoNumber false, DBAccessibleFromOPCUA true, IsOnlyStoredInLoadMemory false, IsWriteProtectedInAS false
   VAR
      Time_Local_read : DTL;
      Time_System_read : DTL;
      Time_System_write : DTL;
      zegar : Time_Of_Day;
   END_VAR
BEGIN
END_DATA_BLOCK

DATA_BLOCK "Czasy pracy DM"   // DB30
{ S7_Optimized_Access := 'FALSE' }
VERSION : 0.1
// stored: AutoNumber false, DBAccessibleFromOPCUA true, IsOnlyStoredInLoadMemory false, IsWriteProtectedInAS false
   VAR
      Sek_P1 : Int := 1;   // Licznik sekund
      Sek_P2 : Int := 2;   // Licznik sekund
      Sek_P3 : Int := 3;   // Licznik sekund
      Sek_P4 : Int := 3;
      Edge_P1 : Bool;   // Pamięć zbocza
      Edge_P2 : Bool;   // Pamięć zbocza
      Edge_P3 : Bool;   // Pamięć zbocza
      Edge_P4 : Bool := false;
      Sek_a : Int;   // Licznik sekund
      Sek_b : Int;   // Licznik sekund
      Edge_a : Bool;   // Pamięć zbocza
      Edge_b : Bool;   // Pamięć zbocza
      Sum_sek_hur_P1 : Real;   // Licznik sumator godzin i sekund na potrzeby wyznaczania dumchawy do pracy
      Sum_sek_hur_P2 : Real := 0.0;   // Licznik sumator godzin i sekund na potrzeby wyznaczania dumchawy do pracy
      Sum_sek_hur_P3 : Real := 0.0;   // Licznik sumator godzin i sekund na potrzeby wyznaczania dumchawy do pracy
      Sum_sek_hur_P4 : Real := 0.0;
   END_VAR
BEGIN
END_DATA_BLOCK

DATA_BLOCK "KALMAN_DB"   // DB125
{ S7_Optimized_Access := 'TRUE' }
VERSION : 0.1
// stored: AutoNumber false, DBAccessibleFromOPCUA true, IsOnlyStoredInLoadMemory false, IsRetainMemResEnabled false, IsWriteProtectedInAS false, MemoryReserve 250
   VAR
      kalman_P : Array[0..4] of Real;
      kalman_K : Array[0..4] of Real;
      kalman_Q : Array[0..4] of Real;
      kalman_R : Array[0..4] of Real;
      kalman_napiecie : Array[0..4] of Real;
      pomiar_napiecie : Array[0..4] of Real;
      wejscie_anal : Array[0..4] of Word;
   END_VAR
BEGIN
   // kalman_napiecie[0] : ciśnienie B6 tłoczenie
   // kalman_napiecie[1] : ciśnienie B7 zasilania
   // kalman_napiecie[2] : ciśnienie B8 ssania
   // kalman_napiecie[3] : przepływ
   // pomiar_napiecie[0] : ciśnienie B6 tłoczenie
   // pomiar_napiecie[1] : ciśnienie B7 zasilania
   // pomiar_napiecie[2] : ciśnienie B8 ssania
   // pomiar_napiecie[3] : przepływ
END_DATA_BLOCK

DATA_BLOCK "dbTable of value Hz"   // DB59
TITLE = Table of value Hz manual instruction
{ S7_Optimized_Access := 'TRUE' }
AUTHOR : rtecmer
VERSION : 0.1
// tabela z wartościami Hz przekazywanymi w instrukcji manualnego sterowania regulatorem PID podczas doączenia kompresora dodatkowego po ustawieniu Set 50Hz
// stored: AutoNumber true, DBAccessibleFromOPCUA true, IsOnlyStoredInLoadMemory false, IsRetainMemResEnabled false, IsWriteProtectedInAS false, MemoryReserve 500
   VAR
      Static_1 : Array[0..20] of Real;
      Static_2 : Array[0..10] of Int;
   END_VAR
BEGIN
   Static_1[0] := 5.0;
   Static_1[1] := 5.3;
   Static_1[2] := 6.0;
   Static_1[3] := 6.7;
   Static_1[4] := 7.2;
   Static_1[5] := 8.0;
   Static_1[6] := 9.0;
   Static_1[7] := 60.0;
   Static_1[8] := 70.0;
   Static_1[9] := 80.0;
   Static_1[10] := 90.0;
   Static_1[11] := 100.0;
   Static_1[12] := 92.0;
   Static_1[13] := 93.0;
   Static_1[14] := 94.0;
   Static_1[15] := 95.0;
   Static_1[16] := 96.0;
   Static_1[17] := 97.0;
   Static_1[18] := 98.0;
   Static_1[19] := 99.0;
   Static_1[20] := 100.0;
   Static_2[0] := 8500;
   Static_2[1] := 9500;
   Static_2[2] := 10000;
   Static_2[3] := 10500;
   Static_2[4] := 11000;
   Static_2[5] := 12000;
   Static_2[6] := 13000;
   Static_2[7] := 19000;
   Static_2[8] := 20500;
   Static_2[9] := 25600;
   Static_2[10] := 27648;
END_DATA_BLOCK

DATA_BLOCK "dbTimersForDrivers"   // DB4
{ S7_Optimized_Access := 'FALSE' }
VERSION : 0.1
// stored: AutoNumber true, DBAccessibleFromOPCUA true, IsOnlyStoredInLoadMemory false, IsWriteProtectedInAS false
   VAR
      TimerP1 { S7_SetPoint := 'True'} : IEC_TIMER;   // Timer drivera
      TimerP2 { S7_SetPoint := 'True'} : IEC_TIMER;   // Timer drivera
      TimerP3 { S7_SetPoint := 'True'} : IEC_TIMER;   // Timer drivera
      ResetModeAut { S7_SetPoint := 'True'} : IEC_TIMER;   // Delay Reset Mode Work Aut
      TimerZ11 { S7_SetPoint := 'True'} : IEC_TIMER;   // Timer drivera Z11
      TimerZ12 { S7_SetPoint := 'True'} : IEC_TIMER;   // Timer drivera Z12
      TimerP4 { S7_SetPoint := 'True'} : IEC_TIMER;   // Timer drivera
      Timer_OFF_Inverter_P1 { S7_SetPoint := 'True'} : IEC_TIMER;   // Timer blokowania dołączenie stycznika falownika P1
      Timer_OFF_Inverter_P2 { S7_SetPoint := 'True'} : IEC_TIMER;   // Timer blokowania dołączenie stycznika falownik P2
      Timer_OFF_Inverter_P3 { S7_SetPoint := 'True'} : IEC_TIMER;   // Timer blokowania dołączenie stycznika falownik P3
      Timer_OFF_Inverter_P4 { S7_SetPoint := 'True'} : IEC_TIMER;   // Timer blokowania dołączenie stycznika falownik P4
      Timer_Start_Network_P1 { S7_SetPoint := 'True'} : IEC_TIMER;   // Timer opóźnienia przełaczenia na sieć
      Timer_Start_Network_P2 { S7_SetPoint := 'True'} : IEC_TIMER;   // Timer opóźnienia przełaczenia na sieć
      Timer_Start_Network_P3 { S7_SetPoint := 'True'} : IEC_TIMER;   // Timer opóźnienia przełaczenia na sieć
      Timer_Start_Network_P4 { S7_SetPoint := 'True'} : IEC_TIMER;   // Timer opóźnienia przełaczenia na sieć
      Timer_Start_Inver_P1 { S7_SetPoint := 'True'} : IEC_TIMER;   // Timer opóźnienia przełaczenia na falownik
      Timer_Start_Inver_P2 { S7_SetPoint := 'True'} : IEC_TIMER;   // Timer opóźnienia przełaczenia na falownik
      Timer_Start_Inver_P3 { S7_SetPoint := 'True'} : IEC_TIMER;   // Timer opóźnienia przełaczenia na falownik
      Timer_Start_Inver_P4 { S7_SetPoint := 'True'} : IEC_TIMER;   // Timer opóźnienia przełaczenia na falownik
      Timer_Hiteresis_On_Set50Hz_Inver_P1 { S7_SetPoint := 'True'} : IEC_TIMER;   // Timer opóźnieniawyłączeniea falownika
      Timer_Hiteresis_On_Set50Hz_Inver_P2 { S7_SetPoint := 'True'} : IEC_TIMER;   // Timer opóźnieniawyłączeniea falownika
      Timer_Hiteresis_On_Set50Hz_Inver_P3 { S7_SetPoint := 'True'} : IEC_TIMER;   // Timer opóźnieniawyłączeniea falownika
      Timer_Hiteresis_On_Set50Hz_Inver_P4 { S7_SetPoint := 'True'} : IEC_TIMER;   // Timer opóźnieniawyłączeniea falownika
      ResetBit_KasowaniaAlarm { S7_SetPoint := 'True'} : IEC_TIMER;   // Timer impulsu kasowania bitu kasowania alarmów HMI
      TimerAlarm_1 { S7_SetPoint := 'True'} : IEC_TIMER;   // Timer impulsu kasowania bitu kasowania alarmów HMI
   END_VAR
BEGIN
   TimerP1.PT := T#10S;
   TimerP2.PT := T#10S;
   TimerP3.PT := T#10S;
   ResetModeAut.PT := T#2S;
   TimerZ11.PT := T#30S;
   TimerZ12.PT := T#30S;
   TimerP4.PT := T#10S;
   Timer_OFF_Inverter_P1.PT := T#5S;
   Timer_OFF_Inverter_P2.PT := T#5S;
   Timer_OFF_Inverter_P3.PT := T#5S;
   Timer_OFF_Inverter_P4.PT := T#5S;
   Timer_Start_Network_P1.PT := T#3S;
   Timer_Start_Network_P2.PT := T#3S;
   Timer_Start_Network_P3.PT := T#3S;
   Timer_Start_Network_P4.PT := T#3S;
   Timer_Start_Inver_P1.PT := T#3100ms;
   Timer_Start_Inver_P2.PT := T#3200ms;
   Timer_Start_Inver_P3.PT := T#3300ms;
   Timer_Start_Inver_P4.PT := T#3400ms;
   Timer_Hiteresis_On_Set50Hz_Inver_P1.PT := T#10ms;
   Timer_Hiteresis_On_Set50Hz_Inver_P2.PT := T#10ms;
   Timer_Hiteresis_On_Set50Hz_Inver_P3.PT := T#10ms;
   Timer_Hiteresis_On_Set50Hz_Inver_P4.PT := T#10ms;
   ResetBit_KasowaniaAlarm.PT := T#2S;
   TimerAlarm_1.PT := T#5M;
END_DATA_BLOCK

